LIN {X 0,Y 537.987,Z 364.092,A -85,B 0,C 180,E1 -4179.8,E2 -4179.8} C_VEL
LIN {X 0,Y 537.969,Z 364.095,A -85,B 0,C 180,E1 -4180.277,E2 -4180.277} C_VEL
LIN {X 0,Y 537.309,Z 364.183,A -85,B 0,C 180,E1 -4180.902,E2 -4180.902} C_VEL
LIN {X 0,Y 534.453,Z 364.538,A -85,B 0,C 180,E1 -4181.917,E2 -4181.917} C_VEL
LIN {X 0,Y 532.034,Z 364.837,A -85,B 0,C 180,E1 -4182.734,E2 -4182.734} C_VEL
LIN {X 0,Y 530.996,Z 364.964,A -85,B 0,C 180,E1 -4183.365,E2 -4183.365} C_VEL
LIN {X 0,Y 530.911,Z 364.973,A -85,B 0,C 180,E1 -4183.578,E2 -4183.578} C_VEL
LIN {X 0,Y 530.912,Z 364.974,A -85,B 0,C 180,E1 -4186.502,E2 -4186.502} C_VEL
LIN {X 0,Y 530.93,Z 364.969,A -85,B 0,C 180,E1 -4189.565,E2 -4189.565} C_VEL
LIN {X 0,Y 530.923,Z 364.975,A -85,B 0,C 180,E1 -4192.584,E2 -4192.584} C_VEL
LIN {X 0,Y 530.957,Z 364.96,A -85,B 0,C 180,E1 -4195.31,E2 -4195.31} C_VEL
LIN {X 0,Y 531.002,Z 365.136,A -85,B 0,C 180,E1 -4197.688,E2 -4197.688} C_VEL
LIN {X 0,Y 535.466,Z 381.503,A -85,B 0,C 180,E1 -4199.65,E2 -4199.65} C_VEL
LIN {X 0,Y 534.889,Z 405.466,A -85,B 0,C 180,E1 -4202.092,E2 -4202.092} C_VEL
LIN {X 0,Y 534.34,Z 429.212,A -85,B 0,C 180,E1 -4204.486,E2 -4204.486} C_VEL
LIN {X 0,Y 533.665,Z 459.976,A -85,B 0,C 180,E1 -4207.55,E2 -4207.55} C_VEL
LIN {X 0,Y 533.378,Z 473.259,A -85,B 0,C 180,E1 -4208.843,E2 -4208.843} C_VEL
LIN {X 0,Y 535.191,Z 484.127,A -85,B 0,C 180,E1 -4209.081,E2 -4209.081} C_VEL
LIN {X 0,Y 534.273,Z 640.741,A -85,B 0,C 180,E1 -4211.258,E2 -4211.258} C_VEL
LIN {X 0,Y 534.016,Z 655.888,A -85,B 0,C 180,E1 -4211.614,E2 -4211.614} C_VEL
LIN {X 0,Y 533.713,Z 669.614,A -85,B 0,C 180,E1 -4212.074,E2 -4212.074} C_VEL
LIN {X 0,Y 533.322,Z 682.934,A -85,B 0,C 180,E1 -4212.655,E2 -4212.655} C_VEL
LIN {X 0,Y 532.901,Z 696.987,A -85,B 0,C 180,E1 -4213.431,E2 -4213.431} C_VEL
LIN {X 0,Y 532.48,Z 710.223,A -85,B 0,C 180,E1 -4214.333,E2 -4214.333} C_VEL
LIN {X 0,Y 532.056,Z 722.77,A -85,B 0,C 180,E1 -4215.369,E2 -4215.369} C_VEL
LIN {X 0,Y 531.65,Z 733.601,A -85,B 0,C 180,E1 -4216.431,E2 -4216.431} C_VEL
LIN {X 0,Y 531.333,Z 743.593,A -85,B 0,C 180,E1 -4217.589,E2 -4217.589} C_VEL
LIN {X 0,Y 531.084,Z 753.363,A -85,B 0,C 180,E1 -4218.939,E2 -4218.939} C_VEL
LIN {X 0,Y 530.801,Z 761.478,A -85,B 0,C 180,E1 -4220.282,E2 -4220.282} C_VEL
LIN {X 0,Y 530.667,Z 768.204,A -85,B 0,C 180,E1 -4221.625,E2 -4221.625} C_VEL
LIN {X 0,Y 530.55,Z 774.441,A -85,B 0,C 180,E1 -4223.154,E2 -4223.154} C_VEL
LIN {X 0,Y 530.508,Z 779.264,A -85,B 0,C 180,E1 -4224.68,E2 -4224.68} C_VEL
LIN {X 0,Y 530.48,Z 782.801,A -85,B 0,C 180,E1 -4226.203,E2 -4226.203} C_VEL
LIN {X 0,Y 530.408,Z 785.143,A -85,B 0,C 180,E1 -4227.723,E2 -4227.723} C_VEL
LIN {X 0,Y 530.34,Z 786.339,A -85,B 0,C 180,E1 -4229.242,E2 -4229.242} C_VEL
LIN {X 0,Y 530.341,Z 786.358,A -85,B 0,C 180,E1 -4230.76,E2 -4230.76} C_VEL
LIN {X 0,Y 530.41,Z 785.237,A -85,B 0,C 180,E1 -4232.279,E2 -4232.279} C_VEL
LIN {X 0,Y 530.482,Z 782.969,A -85,B 0,C 180,E1 -4233.799,E2 -4233.799} C_VEL
LIN {X 0,Y 530.507,Z 779.504,A -85,B 0,C 180,E1 -4235.322,E2 -4235.322} C_VEL
LIN {X 0,Y 530.551,Z 774.76,A -85,B 0,C 180,E1 -4236.848,E2 -4236.848} C_VEL
LIN {X 0,Y 530.661,Z 768.615,A -85,B 0,C 180,E1 -4238.378,E2 -4238.378} C_VEL
LIN {X 0,Y 530.808,Z 760.885,A -85,B 0,C 180,E1 -4239.912,E2 -4239.912} C_VEL
LIN {X 0,Y 531.045,Z 752.644,A -85,B 0,C 180,E1 -4241.258,E2 -4241.258} C_VEL
LIN {X 0,Y 531.356,Z 742.721,A -85,B 0,C 180,E1 -4242.607,E2 -4242.607} C_VEL
LIN {X 0,Y 531.687,Z 732.601,A -85,B 0,C 180,E1 -4243.765,E2 -4243.765} C_VEL
LIN {X 0,Y 532.105,Z 720.489,A -85,B 0,C 180,E1 -4244.926,E2 -4244.926} C_VEL
LIN {X 0,Y 532.562,Z 708.684,A -85,B 0,C 180,E1 -4245.874,E2 -4245.874} C_VEL
LIN {X 0,Y 533.019,Z 695.268,A -85,B 0,C 180,E1 -4246.765,E2 -4246.765} C_VEL
LIN {X 0,Y 533.399,Z 680.725,A -85,B 0,C 180,E1 -4247.543,E2 -4247.543} C_VEL
LIN {X 0,Y 533.769,Z 666.821,A -85,B 0,C 180,E1 -4248.124,E2 -4248.124} C_VEL
LIN {X 0,Y 534.11,Z 651.426,A -85,B 0,C 180,E1 -4248.6,E2 -4248.6} C_VEL
LIN {X 0,Y 534.346,Z 635.503,A -85,B 0,C 180,E1 -4248.923,E2 -4248.923} C_VEL
LIN {X 0,Y 535.19,Z 484.115,A -85,B 0,C 180,E1 -4251.009,E2 -4251.009} C_VEL
LIN {X 0,Y 533.363,Z 472.907,A -85,B 0,C 180,E1 -4251.269,E2 -4251.269} C_VEL
LIN {X 0,Y 533.98,Z 444.484,A -85,B 0,C 180,E1 -4254.081,E2 -4254.081} C_VEL
LIN {X 0,Y 534.661,Z 417.063,A -85,B 0,C 180,E1 -4256.822,E2 -4256.822} C_VEL
LIN {X 0,Y 535.33,Z 389.185,A -85,B 0,C 180,E1 -4259.654,E2 -4259.654} C_VEL
LIN {X 0,Y 535.433,Z 381.261,A -85,B 0,C 180,E1 -4260.464,E2 -4260.464} C_VEL
LIN {X 0,Y 530.964,Z 365.143,A -85,B 0,C 180,E1 -4262.406,E2 -4262.406} C_VEL
LIN {X 0,Y 530.911,Z 364.972,A -85,B 0,C 180,E1 -4264.842,E2 -4264.842} C_VEL
LIN {X 0,Y 530.901,Z 364.981,A -85,B 0,C 180,E1 -4267.514,E2 -4267.514} C_VEL
LIN {X 0,Y 530.908,Z 364.975,A -85,B 0,C 180,E1 -4270.441,E2 -4270.441} C_VEL
LIN {X 0,Y 530.922,Z 364.977,A -85,B 0,C 180,E1 -4273.5,E2 -4273.5} C_VEL
LIN {X 0,Y 530.962,Z 364.966,A -85,B 0,C 180,E1 -4275.625,E2 -4275.625} C_VEL
LIN {X 0,Y 530.913,Z 364.975,A -85,B 0,C 180,E1 -4278.557,E2 -4278.557} C_VEL
LIN {X 0,Y 530.931,Z 364.975,A -85,B 0,C 180,E1 -4281.527,E2 -4281.527} C_VEL
LIN {X 0,Y 530.931,Z 364.967,A -85,B 0,C 180,E1 -4284.378,E2 -4284.378} C_VEL
LIN {X 0,Y 530.948,Z 364.972,A -85,B 0,C 180,E1 -4287.132,E2 -4287.132} C_VEL
LIN {X 0,Y 530.936,Z 364.971,A -85,B 0,C 180,E1 -4289.801,E2 -4289.801} C_VEL
LIN {X 0,Y 530.958,Z 364.969,A -85,B 0,C 180,E1 -4292.48,E2 -4292.48} C_VEL
LIN {X 0,Y 530.95,Z 364.971,A -85,B 0,C 180,E1 -4295.774,E2 -4295.774} C_VEL
LIN {X 0,Y 530.999,Z 364.97,A -85,B 0,C 180,E1 -4299.062,E2 -4299.062} C_VEL
LIN {X 0,Y 531.055,Z 365.122,A -85,B 0,C 180,E1 -4299.647,E2 -4299.647} C_VEL
LIN {X 0,Y 532.05,Z 371.983,A -85,B 0,C 180,E1 -4300.917,E2 -4300.917} C_VEL
LIN {X 0,Y 531.965,Z 377.818,A -85,B 0,C 180,E1 -4301.904,E2 -4301.904} C_VEL
LIN {X 0,Y 533.976,Z 387.187,A -85,B 0,C 180,E1 -4302.145,E2 -4302.145} C_VEL
LIN {X 0,Y 533.214,Z 515.389,A -85,B 0,C 180,E1 -4303.985,E2 -4303.985} C_VEL
LIN {X 0,Y 533.039,Z 529.891,A -85,B 0,C 180,E1 -4304.355,E2 -4304.355} C_VEL
LIN {X 0,Y 532.821,Z 543.338,A -85,B 0,C 180,E1 -4304.851,E2 -4304.851} C_VEL
LIN {X 0,Y 532.614,Z 556.223,A -85,B 0,C 180,E1 -4305.48,E2 -4305.48} C_VEL
LIN {X 0,Y 532.292,Z 567.295,A -85,B 0,C 180,E1 -4306.154,E2 -4306.154} C_VEL
LIN {X 0,Y 531.981,Z 578.921,A -85,B 0,C 180,E1 -4307.021,E2 -4307.021} C_VEL
LIN {X 0,Y 531.662,Z 589.877,A -85,B 0,C 180,E1 -4308.017,E2 -4308.017} C_VEL
LIN {X 0,Y 531.433,Z 599.998,A -85,B 0,C 180,E1 -4309.138,E2 -4309.138} C_VEL
LIN {X 0,Y 531.15,Z 608.633,A -85,B 0,C 180,E1 -4310.287,E2 -4310.287} C_VEL
LIN {X 0,Y 530.914,Z 616.868,A -85,B 0,C 180,E1 -4311.627,E2 -4311.627} C_VEL
LIN {X 0,Y 530.781,Z 622.612,A -85,B 0,C 180,E1 -4312.774,E2 -4312.774} C_VEL
LIN {X 0,Y 530.724,Z 628.655,A -85,B 0,C 180,E1 -4314.3,E2 -4314.3} C_VEL
LIN {X 0,Y 530.61,Z 632.169,A -85,B 0,C 180,E1 -4315.442,E2 -4315.442} C_VEL
LIN {X 0,Y 530.578,Z 635.531,A -85,B 0,C 180,E1 -4316.963,E2 -4316.963} C_VEL
LIN {X 0,Y 530.475,Z 637.559,A -85,B 0,C 180,E1 -4318.482,E2 -4318.482} C_VEL
LIN {X 0,Y 530.478,Z 638.29,A -85,B 0,C 180,E1 -4320,E2 -4320} C_VEL
LIN {X 0,Y 530.475,Z 637.723,A -85,B 0,C 180,E1 -4321.518,E2 -4321.518} C_VEL
LIN {X 0,Y 530.595,Z 635.831,A -85,B 0,C 180,E1 -4323.037,E2 -4323.037} C_VEL
LIN {X 0,Y 530.631,Z 632.609,A -85,B 0,C 180,E1 -4324.558,E2 -4324.558} C_VEL
LIN {X 0,Y 530.785,Z 627.929,A -85,B 0,C 180,E1 -4326.08,E2 -4326.08} C_VEL
LIN {X 0,Y 530.864,Z 621.641,A -85,B 0,C 180,E1 -4327.608,E2 -4327.608} C_VEL
LIN {X 0,Y 531.068,Z 614.585,A -85,B 0,C 180,E1 -4328.945,E2 -4328.945} C_VEL
LIN {X 0,Y 531.304,Z 605.793,A -85,B 0,C 180,E1 -4330.287,E2 -4330.287} C_VEL
LIN {X 0,Y 531.601,Z 596.53,A -85,B 0,C 180,E1 -4331.438,E2 -4331.438} C_VEL
LIN {X 0,Y 531.887,Z 586.212,A -85,B 0,C 180,E1 -4332.496,E2 -4332.496} C_VEL
LIN {X 0,Y 532.236,Z 574.76,A -85,B 0,C 180,E1 -4333.458,E2 -4333.458} C_VEL
LIN {X 0,Y 532.459,Z 563.55,A -85,B 0,C 180,E1 -4334.231,E2 -4334.231} C_VEL
LIN {X 0,Y 532.774,Z 551.386,A -85,B 0,C 180,E1 -4334.906,E2 -4334.906} C_VEL
LIN {X 0,Y 533.05,Z 539.454,A -85,B 0,C 180,E1 -4335.427,E2 -4335.427} C_VEL
LIN {X 0,Y 533.129,Z 525.988,A -85,B 0,C 180,E1 -4335.87,E2 -4335.87} C_VEL
LIN {X 0,Y 533.254,Z 510.983,A -85,B 0,C 180,E1 -4336.19,E2 -4336.19} C_VEL
LIN {X 0,Y 534.274,Z 387.61,A -85,B 0,C 180,E1 -4338.018,E2 -4338.018} C_VEL
LIN {X 0,Y 532.643,Z 380.641,A -85,B 0,C 180,E1 -4338.214,E2 -4338.214} C_VEL
LIN {X 0,Y 532.776,Z 373.678,A -85,B 0,C 180,E1 -4339.456,E2 -4339.456} C_VEL
LIN {X 0,Y 531.009,Z 365.099,A -85,B 0,C 180,E1 -4341.191,E2 -4341.191} C_VEL
LIN {X 0,Y 530.975,Z 364.971,A -85,B 0,C 180,E1 -4344.225,E2 -4344.225} C_VEL
LIN {X 0,Y 531.005,Z 364.969,A -85,B 0,C 180,E1 -4346.744,E2 -4346.744} C_VEL
LIN {X 0,Y 530.986,Z 364.967,A -85,B 0,C 180,E1 -4349.322,E2 -4349.322} C_VEL
LIN {X 0,Y 530.97,Z 364.971,A -85,B 0,C 180,E1 -4352.1,E2 -4352.1} C_VEL
LIN {X 0,Y 530.973,Z 364.971,A -85,B 0,C 180,E1 -4354.85,E2 -4354.85} C_VEL
LIN {X 0,Y 530.967,Z 364.968,A -85,B 0,C 180,E1 -4357.507,E2 -4357.507} C_VEL
LIN {X 0,Y 530.984,Z 364.972,A -85,B 0,C 180,E1 -4360.433,E2 -4360.433} C_VEL
LIN {X 0,Y 530.936,Z 364.971,A -85,B 0,C 180,E1 -4363.277,E2 -4363.277} C_VEL
LIN {X 0,Y 530.973,Z 364.969,A -85,B 0,C 180,E1 -4365.622,E2 -4365.622} C_VEL
LIN {X 0,Y 530.963,Z 364.972,A -85,B 0,C 180,E1 -4368.561,E2 -4368.561} C_VEL
LIN {X 0,Y 530.952,Z 364.973,A -85,B 0,C 180,E1 -4371.528,E2 -4371.528} C_VEL
LIN {X 0,Y 530.93,Z 364.977,A -85,B 0,C 180,E1 -4374.377,E2 -4374.377} C_VEL
LIN {X 0,Y 530.947,Z 364.974,A -85,B 0,C 180,E1 -4377.131,E2 -4377.131} C_VEL
LIN {X 0,Y 530.976,Z 365.169,A -85,B 0,C 180,E1 -4378.755,E2 -4378.755} C_VEL
LIN {X 0,Y 533.789,Z 375.588,A -85,B 0,C 180,E1 -4379.978,E2 -4379.978} C_VEL
LIN {X 0,Y 535.109,Z 381.227,A -85,B 0,C 180,E1 -4380.596,E2 -4380.596} C_VEL
LIN {X 0,Y 534.431,Z 411.488,A -85,B 0,C 180,E1 -4383.44,E2 -4383.44} C_VEL
LIN {X 0,Y 533.737,Z 445.316,A -85,B 0,C 180,E1 -4386.526,E2 -4386.526} C_VEL
LIN {X 0,Y 533.232,Z 471.07,A -85,B 0,C 180,E1 -4388.824,E2 -4388.824} C_VEL
LIN {X 0,Y 535.077,Z 484.407,A -85,B 0,C 180,E1 -4389.096,E2 -4389.096} C_VEL
LIN {X 0,Y 534.169,Z 640.097,A -85,B 0,C 180,E1 -4391.243,E2 -4391.243} C_VEL
LIN {X 0,Y 533.929,Z 655.851,A -85,B 0,C 180,E1 -4391.608,E2 -4391.608} C_VEL
LIN {X 0,Y 533.612,Z 671.04,A -85,B 0,C 180,E1 -4392.118,E2 -4392.118} C_VEL
LIN {X 0,Y 533.297,Z 685.298,A -85,B 0,C 180,E1 -4392.751,E2 -4392.751} C_VEL
LIN {X 0,Y 532.825,Z 699.152,A -85,B 0,C 180,E1 -4393.525,E2 -4393.525} C_VEL
LIN {X 0,Y 532.444,Z 711.668,A -85,B 0,C 180,E1 -4394.398,E2 -4394.398} C_VEL
LIN {X 0,Y 531.968,Z 724.282,A -85,B 0,C 180,E1 -4395.461,E2 -4395.461} C_VEL
LIN {X 0,Y 531.609,Z 735.737,A -85,B 0,C 180,E1 -4396.622,E2 -4396.622} C_VEL
LIN {X 0,Y 531.288,Z 745.38,A -85,B 0,C 180,E1 -4397.78,E2 -4397.78} C_VEL
LIN {X 0,Y 531.042,Z 754.844,A -85,B 0,C 180,E1 -4399.128,E2 -4399.128} C_VEL
LIN {X 0,Y 530.765,Z 762.723,A -85,B 0,C 180,E1 -4400.472,E2 -4400.472} C_VEL
LIN {X 0,Y 530.641,Z 770.083,A -85,B 0,C 180,E1 -4402.005,E2 -4402.005} C_VEL
LIN {X 0,Y 530.522,Z 775.774,A -85,B 0,C 180,E1 -4403.488,E2 -4403.488} C_VEL
LIN {X 0,Y 530.508,Z 779.383,A -85,B 0,C 180,E1 -4404.678,E2 -4404.678} C_VEL
LIN {X 0,Y 530.481,Z 782.881,A -85,B 0,C 180,E1 -4406.201,E2 -4406.201} C_VEL
LIN {X 0,Y 530.407,Z 785.185,A -85,B 0,C 180,E1 -4407.721,E2 -4407.721} C_VEL
LIN {X 0,Y 530.341,Z 786.347,A -85,B 0,C 180,E1 -4409.24,E2 -4409.24} C_VEL
LIN {X 0,Y 530.341,Z 786.348,A -85,B 0,C 180,E1 -4410.758,E2 -4410.758} C_VEL
LIN {X 0,Y 530.407,Z 785.191,A -85,B 0,C 180,E1 -4412.277,E2 -4412.277} C_VEL
LIN {X 0,Y 530.48,Z 782.889,A -85,B 0,C 180,E1 -4413.797,E2 -4413.797} C_VEL
LIN {X 0,Y 530.508,Z 779.389,A -85,B 0,C 180,E1 -4415.32,E2 -4415.32} C_VEL
LIN {X 0,Y 530.548,Z 774.61,A -85,B 0,C 180,E1 -4416.846,E2 -4416.846} C_VEL
LIN {X 0,Y 530.664,Z 768.428,A -85,B 0,C 180,E1 -4418.375,E2 -4418.375} C_VEL
LIN {X 0,Y 530.818,Z 760.655,A -85,B 0,C 180,E1 -4419.91,E2 -4419.91} C_VEL
LIN {X 0,Y 531.055,Z 752.376,A -85,B 0,C 180,E1 -4421.255,E2 -4421.255} C_VEL
LIN {X 0,Y 531.38,Z 742.401,A -85,B 0,C 180,E1 -4422.604,E2 -4422.604} C_VEL
LIN {X 0,Y 531.708,Z 732.196,A -85,B 0,C 180,E1 -4423.762,E2 -4423.762} C_VEL
LIN {X 0,Y 532.118,Z 720.025,A -85,B 0,C 180,E1 -4424.923,E2 -4424.923} C_VEL
LIN {X 0,Y 532.6,Z 706.602,A -85,B 0,C 180,E1 -4425.979,E2 -4425.979} C_VEL
LIN {X 0,Y 532.98,Z 694.363,A -85,B 0,C 180,E1 -4426.764,E2 -4426.764} C_VEL
LIN {X 0,Y 533.408,Z 679.29,A -85,B 0,C 180,E1 -4427.54,E2 -4427.54} C_VEL
LIN {X 0,Y 533.779,Z 664.666,A -85,B 0,C 180,E1 -4428.122,E2 -4428.122} C_VEL
LIN {X 0,Y 534.089,Z 648.748,A -85,B 0,C 180,E1 -4428.586,E2 -4428.586} C_VEL
LIN {X 0,Y 534.281,Z 632.911,A -85,B 0,C 180,E1 -4428.882,E2 -4428.882} C_VEL
LIN {X 0,Y 535.114,Z 484.112,A -85,B 0,C 180,E1 -4430.922,E2 -4430.922} C_VEL
LIN {X 0,Y 533.337,Z 471.527,A -85,B 0,C 180,E1 -4431.194,E2 -4431.194} C_VEL
LIN {X 0,Y 534.024,Z 441.043,A -85,B 0,C 180,E1 -4433.973,E2 -4433.973} C_VEL
LIN {X 0,Y 534.894,Z 407.916,A -85,B 0,C 180,E1 -4437.059,E2 -4437.059} C_VEL
LIN {X 0,Y 535.563,Z 383.049,A -85,B 0,C 180,E1 -4439.427,E2 -4439.427} C_VEL
LIN {X 0,Y 535.511,Z 381.106,A -85,B 0,C 180,E1 -4439.622,E2 -4439.622} C_VEL
LIN {X 0,Y 530.983,Z 365.172,A -85,B 0,C 180,E1 -4441.492,E2 -4441.492} C_VEL
LIN {X 0,Y 530.94,Z 364.976,A -85,B 0,C 180,E1 -4443.774,E2 -4443.774} C_VEL
LIN {X 0,Y 530.896,Z 364.98,A -85,B 0,C 180,E1 -4446.561,E2 -4446.561} C_VEL
LIN {X 0,Y 530.955,Z 364.969,A -85,B 0,C 180,E1 -4449.444,E2 -4449.444} C_VEL
LIN {X 0,Y 530.919,Z 364.98,A -85,B 0,C 180,E1 -4452.46,E2 -4452.46} C_VEL
LIN {X 0,Y 530.947,Z 364.968,A -85,B 0,C 180,E1 -4455.449,E2 -4455.449} C_VEL
LIN {X 0,Y 530.938,Z 364.967,A -85,B 0,C 180,E1 -4458.559,E2 -4458.559} C_VEL
LIN {X 0,Y 530.934,Z 364.97,A -85,B 0,C 180,E1 -4461.527,E2 -4461.527} C_VEL
LIN {X 0,Y 530.915,Z 364.964,A -85,B 0,C 180,E1 -4464.377,E2 -4464.377} C_VEL
LIN {X 0,Y 530.951,Z 364.967,A -85,B 0,C 180,E1 -4467.132,E2 -4467.132} C_VEL
LIN {X 0,Y 530.934,Z 364.971,A -85,B 0,C 180,E1 -4469.801,E2 -4469.801} C_VEL
LIN {X 0,Y 530.946,Z 364.977,A -85,B 0,C 180,E1 -4472.478,E2 -4472.478} C_VEL
LIN {X 0,Y 530.937,Z 364.967,A -85,B 0,C 180,E1 -4474.939,E2 -4474.939} C_VEL
LIN {X 0,Y 530.96,Z 364.968,A -85,B 0,C 180,E1 -4477.898,E2 -4477.898} C_VEL
LIN {X 0,Y 530.952,Z 364.973,A -85,B 0,C 180,E1 -4480.676,E2 -4480.676} C_VEL
LIN {X 0,Y 530.911,Z 364.973,A -85,B 0,C 180,E1 -4483.069,E2 -4483.069} C_VEL
LIN {X 0,Y 530.984,Z 364.959,A -85,B 0,C 180,E1 -4485.435,E2 -4485.435} C_VEL
LIN {X 0,Y 531.013,Z 364.966,A -85,B 0,C 180,E1 -4488.549,E2 -4488.549} C_VEL
LIN {X 0,Y 530.976,Z 364.962,A -85,B 0,C 180,E1 -4491.628,E2 -4491.628} C_VEL
LIN {X 0,Y 531.067,Z 364.955,A -85,B 0,C 180,E1 -4494.685,E2 -4494.685} C_VEL
LIN {X 0,Y 531.108,Z 364.947,A -85,B 0,C 180,E1 -4497.725,E2 -4497.725} C_VEL
LIN {X 0,Y 531.133,Z 364.946,A -85,B 0,C 180,E1 -4500.758,E2 -4500.758} C_VEL
LIN {X 0,Y 531.069,Z 364.956,A -85,B 0,C 180,E1 -4503.034,E2 -4503.034} C_VEL
LIN {X 0,Y 531.029,Z 364.958,A -85,B 0,C 180,E1 -4506.078,E2 -4506.078} C_VEL
LIN {X 0,Y 530.972,Z 364.968,A -85,B 0,C 180,E1 -4508.372,E2 -4508.372} C_VEL
LIN {X 0,Y 531.03,Z 364.952,A -85,B 0,C 180,E1 -4511.67,E2 -4511.67} C_VEL
LIN {X 0,Y 531.006,Z 364.963,A -85,B 0,C 180,E1 -4514.953,E2 -4514.953} C_VEL
LIN {X 0,Y 530.964,Z 364.964,A -85,B 0,C 180,E1 -4517.724,E2 -4517.724} C_VEL
LIN {X 0,Y 531.009,Z 364.961,A -85,B 0,C 180,E1 -4520.128,E2 -4520.128} C_VEL
LIN {X 0,Y 530.926,Z 364.976,A -85,B 0,C 180,E1 -4522.574,E2 -4522.574} C_VEL
LIN {X 0,Y 530.927,Z 364.972,A -85,B 0,C 180,E1 -4525.062,E2 -4525.062} C_VEL
LIN {X 0,Y 530.942,Z 364.969,A -85,B 0,C 180,E1 -4527.6,E2 -4527.6} C_VEL
LIN {X 0,Y 530.93,Z 364.977,A -85,B 0,C 180,E1 -4530.64,E2 -4530.64} C_VEL
LIN {X 0,Y 530.948,Z 364.969,A -85,B 0,C 180,E1 -4533.501,E2 -4533.501} C_VEL
LIN {X 0,Y 530.921,Z 364.972,A -85,B 0,C 180,E1 -4536.153,E2 -4536.153} C_VEL
LIN {X 0,Y 530.944,Z 364.968,A -85,B 0,C 180,E1 -4538.653,E2 -4538.653} C_VEL
LIN {X 0,Y 530.939,Z 364.967,A -85,B 0,C 180,E1 -4541.441,E2 -4541.441} C_VEL
LIN {X 0,Y 530.911,Z 364.973,A -85,B 0,C 180,E1 -4543.578,E2 -4543.578} C_VEL
LIN {X 0,Y 530.249,Z 365.057,A -85,B 0,C 180,E1 -4544.212,E2 -4544.212} C_VEL
LIN {X 0,Y 527.407,Z 365.412,A -85,B 0,C 180,E1 -4545.241,E2 -4545.241} C_VEL
LIN {X 0,Y 524.997,Z 365.712,A -85,B 0,C 180,E1 -4546.07,E2 -4546.07} C_VEL
LIN {X 0,Y 523.953,Z 365.84,A -85,B 0,C 180,E1 -4546.709,E2 -4546.709} C_VEL
LIN {X 0,Y 523.862,Z 365.851,A -85,B 0,C 180,E1 -4546.926,E2 -4546.926} C_VEL
LIN {X 0,Y 523.903,Z 365.844,A -85,B 0,C 180,E1 -4549.919,E2 -4549.919} C_VEL
LIN {X 0,Y 523.864,Z 365.852,A -85,B 0,C 180,E1 -4552.866,E2 -4552.866} C_VEL
LIN {X 0,Y 523.901,Z 365.832,A -85,B 0,C 180,E1 -4555.709,E2 -4555.709} C_VEL
LIN {X 0,Y 523.961,Z 366.063,A -85,B 0,C 180,E1 -4557.383,E2 -4557.383} C_VEL
LIN {X 0,Y 528.709,Z 383.052,A -85,B 0,C 180,E1 -4559.441,E2 -4559.441} C_VEL
LIN {X 0,Y 528.312,Z 403.383,A -85,B 0,C 180,E1 -4561.544,E2 -4561.544} C_VEL
LIN {X 0,Y 527.591,Z 429.824,A -85,B 0,C 180,E1 -4564.242,E2 -4564.242} C_VEL
LIN {X 0,Y 526.883,Z 458.525,A -85,B 0,C 180,E1 -4567.125,E2 -4567.125} C_VEL
LIN {X 0,Y 526.559,Z 472.845,A -85,B 0,C 180,E1 -4568.536,E2 -4568.536} C_VEL
LIN {X 0,Y 528.621,Z 486.323,A -85,B 0,C 180,E1 -4568.841,E2 -4568.841} C_VEL
LIN {X 0,Y 527.557,Z 640.53,A -85,B 0,C 180,E1 -4571.008,E2 -4571.008} C_VEL
LIN {X 0,Y 527.286,Z 655.836,A -85,B 0,C 180,E1 -4571.371,E2 -4571.371} C_VEL
LIN {X 0,Y 526.92,Z 670.811,A -85,B 0,C 180,E1 -4571.886,E2 -4571.886} C_VEL
LIN {X 0,Y 526.46,Z 684.812,A -85,B 0,C 180,E1 -4572.522,E2 -4572.522} C_VEL
LIN {X 0,Y 525.998,Z 698.494,A -85,B 0,C 180,E1 -4573.307,E2 -4573.307} C_VEL
LIN {X 0,Y 525.543,Z 711.522,A -85,B 0,C 180,E1 -4574.225,E2 -4574.225} C_VEL
LIN {X 0,Y 525.08,Z 723.802,A -85,B 0,C 180,E1 -4575.269,E2 -4575.269} C_VEL
LIN {X 0,Y 524.631,Z 735.342,A -85,B 0,C 180,E1 -4576.443,E2 -4576.443} C_VEL
LIN {X 0,Y 524.242,Z 746.435,A -85,B 0,C 180,E1 -4577.799,E2 -4577.799} C_VEL
LIN {X 0,Y 523.991,Z 755.799,A -85,B 0,C 180,E1 -4579.178,E2 -4579.178} C_VEL
LIN {X 0,Y 523.746,Z 762.523,A -85,B 0,C 180,E1 -4580.345,E2 -4580.345} C_VEL
LIN {X 0,Y 523.565,Z 769.921,A -85,B 0,C 180,E1 -4581.899,E2 -4581.899} C_VEL
LIN {X 0,Y 523.411,Z 776.044,A -85,B 0,C 180,E1 -4583.526,E2 -4583.526} C_VEL
LIN {X 0,Y 523.441,Z 779.265,A -85,B 0,C 180,E1 -4584.608,E2 -4584.608} C_VEL
LIN {X 0,Y 523.402,Z 782.802,A -85,B 0,C 180,E1 -4586.152,E2 -4586.152} C_VEL
LIN {X 0,Y 523.332,Z 785.143,A -85,B 0,C 180,E1 -4587.692,E2 -4587.692} C_VEL
LIN {X 0,Y 523.246,Z 786.339,A -85,B 0,C 180,E1 -4589.232,E2 -4589.232} C_VEL
LIN {X 0,Y 523.247,Z 786.358,A -85,B 0,C 180,E1 -4590.771,E2 -4590.771} C_VEL
LIN {X 0,Y 523.333,Z 785.237,A -85,B 0,C 180,E1 -4592.31,E2 -4592.31} C_VEL
LIN {X 0,Y 523.403,Z 782.968,A -85,B 0,C 180,E1 -4593.851,E2 -4593.851} C_VEL
LIN {X 0,Y 523.439,Z 779.502,A -85,B 0,C 180,E1 -4595.394,E2 -4595.394} C_VEL
LIN {X 0,Y 523.483,Z 774.756,A -85,B 0,C 180,E1 -4596.941,E2 -4596.941} C_VEL
LIN {X 0,Y 523.609,Z 768.61,A -85,B 0,C 180,E1 -4598.492,E2 -4598.492} C_VEL
LIN {X 0,Y 523.776,Z 760.88,A -85,B 0,C 180,E1 -4600.047,E2 -4600.047} C_VEL
LIN {X 0,Y 524.009,Z 752.637,A -85,B 0,C 180,E1 -4601.411,E2 -4601.411} C_VEL
LIN {X 0,Y 524.365,Z 742.711,A -85,B 0,C 180,E1 -4602.777,E2 -4602.777} C_VEL
LIN {X 0,Y 524.743,Z 732.583,A -85,B 0,C 180,E1 -4603.951,E2 -4603.951} C_VEL
LIN {X 0,Y 525.201,Z 720.559,A -85,B 0,C 180,E1 -4605.118,E2 -4605.118} C_VEL
LIN {X 0,Y 525.683,Z 708.377,A -85,B 0,C 180,E1 -4606.107,E2 -4606.107} C_VEL
LIN {X 0,Y 526.207,Z 695.221,A -85,B 0,C 180,E1 -4606.988,E2 -4606.988} C_VEL
LIN {X 0,Y 526.539,Z 682.661,A -85,B 0,C 180,E1 -4607.678,E2 -4607.678} C_VEL
LIN {X 0,Y 526.977,Z 668.007,A -85,B 0,C 180,E1 -4608.316,E2 -4608.316} C_VEL
LIN {X 0,Y 527.332,Z 652.493,A -85,B 0,C 180,E1 -4608.816,E2 -4608.816} C_VEL
LIN {X 0,Y 527.593,Z 637.697,A -85,B 0,C 180,E1 -4609.134,E2 -4609.134} C_VEL
LIN {X 0,Y 528.572,Z 485.348,A -85,B 0,C 180,E1 -4611.264,E2 -4611.264} C_VEL
LIN {X 0,Y 526.605,Z 473.206,A -85,B 0,C 180,E1 -4611.533,E2 -4611.533} C_VEL
LIN {X 0,Y 527.235,Z 444.14,A -85,B 0,C 180,E1 -4614.409,E2 -4614.409} C_VEL
LIN {X 0,Y 527.954,Z 416.184,A -85,B 0,C 180,E1 -4617.233,E2 -4617.233} C_VEL
LIN {X 0,Y 528.788,Z 386.926,A -85,B 0,C 180,E1 -4620.243,E2 -4620.243} C_VEL
LIN {X 0,Y 528.628,Z 382.804,A -85,B 0,C 180,E1 -4620.677,E2 -4620.677} C_VEL
LIN {X 0,Y 523.925,Z 366.076,A -85,B 0,C 180,E1 -4622.707,E2 -4622.707} C_VEL
LIN {X 0,Y 523.857,Z 365.835,A -85,B 0,C 180,E1 -4623.717,E2 -4623.717} C_VEL
LIN {X 0,Y 523.849,Z 365.854,A -85,B 0,C 180,E1 -4626.393,E2 -4626.393} C_VEL
LIN {X 0,Y 523.888,Z 365.85,A -85,B 0,C 180,E1 -4629.089,E2 -4629.089} C_VEL
LIN {X 0,Y 523.888,Z 365.843,A -85,B 0,C 180,E1 -4632.126,E2 -4632.126} C_VEL
LIN {X 0,Y 523.931,Z 365.842,A -85,B 0,C 180,E1 -4635.312,E2 -4635.312} C_VEL
LIN {X 0,Y 523.883,Z 365.852,A -85,B 0,C 180,E1 -4638.7,E2 -4638.7} C_VEL
LIN {X 0,Y 523.89,Z 365.849,A -85,B 0,C 180,E1 -4641.896,E2 -4641.896} C_VEL
LIN {X 0,Y 523.916,Z 365.841,A -85,B 0,C 180,E1 -4644.914,E2 -4644.914} C_VEL
LIN {X 0,Y 523.903,Z 365.848,A -85,B 0,C 180,E1 -4647.686,E2 -4647.686} C_VEL
LIN {X 0,Y 523.934,Z 365.845,A -85,B 0,C 180,E1 -4650.682,E2 -4650.682} C_VEL
LIN {X 0,Y 523.885,Z 365.851,A -85,B 0,C 180,E1 -4653.724,E2 -4653.724} C_VEL
LIN {X 0,Y 523.911,Z 365.847,A -85,B 0,C 180,E1 -4656.269,E2 -4656.269} C_VEL
LIN {X 0,Y 523.992,Z 365.907,A -85,B 0,C 180,E1 -4659.411,E2 -4659.411} C_VEL
LIN {X 0,Y 525.156,Z 373.557,A -85,B 0,C 180,E1 -4660.86,E2 -4660.86} C_VEL
LIN {X 0,Y 525.09,Z 378.407,A -85,B 0,C 180,E1 -4661.662,E2 -4661.662} C_VEL
LIN {X 0,Y 527.233,Z 388.321,A -85,B 0,C 180,E1 -4661.914,E2 -4661.914} C_VEL
LIN {X 0,Y 526.405,Z 516.027,A -85,B 0,C 180,E1 -4663.788,E2 -4663.788} C_VEL
LIN {X 0,Y 526.229,Z 530.054,A -85,B 0,C 180,E1 -4664.147,E2 -4664.147} C_VEL
LIN {X 0,Y 525.986,Z 543.668,A -85,B 0,C 180,E1 -4664.649,E2 -4664.649} C_VEL
LIN {X 0,Y 525.768,Z 556.66,A -85,B 0,C 180,E1 -4665.287,E2 -4665.287} C_VEL
LIN {X 0,Y 525.424,Z 567.816,A -85,B 0,C 180,E1 -4665.969,E2 -4665.969} C_VEL
LIN {X 0,Y 525.11,Z 579.51,A -85,B 0,C 180,E1 -4666.848,E2 -4666.848} C_VEL
LIN {X 0,Y 524.752,Z 590.726,A -85,B 0,C 180,E1 -4667.876,E2 -4667.876} C_VEL
LIN {X 0,Y 524.509,Z 600.721,A -85,B 0,C 180,E1 -4668.992,E2 -4668.992} C_VEL
LIN {X 0,Y 524.192,Z 609.405,A -85,B 0,C 180,E1 -4670.157,E2 -4670.157} C_VEL
LIN {X 0,Y 523.941,Z 617.704,A -85,B 0,C 180,E1 -4671.515,E2 -4671.515} C_VEL
LIN {X 0,Y 523.793,Z 623.469,A -85,B 0,C 180,E1 -4672.677,E2 -4672.677} C_VEL
LIN {X 0,Y 523.724,Z 629.574,A -85,B 0,C 180,E1 -4674.224,E2 -4674.224} C_VEL
LIN {X 0,Y 523.591,Z 633.102,A -85,B 0,C 180,E1 -4675.381,E2 -4675.381} C_VEL
LIN {X 0,Y 523.555,Z 636.516,A -85,B 0,C 180,E1 -4676.922,E2 -4676.922} C_VEL
LIN {X 0,Y 523.459,Z 638.568,A -85,B 0,C 180,E1 -4678.461,E2 -4678.461} C_VEL
LIN {X 0,Y 523.473,Z 639.314,A -85,B 0,C 180,E1 -4680,E2 -4680} C_VEL
LIN {X 0,Y 523.46,Z 638.762,A -85,B 0,C 180,E1 -4681.539,E2 -4681.539} C_VEL
LIN {X 0,Y 523.581,Z 636.878,A -85,B 0,C 180,E1 -4683.078,E2 -4683.078} C_VEL
LIN {X 0,Y 523.626,Z 633.656,A -85,B 0,C 180,E1 -4684.619,E2 -4684.619} C_VEL
LIN {X 0,Y 523.81,Z 628.953,A -85,B 0,C 180,E1 -4686.162,E2 -4686.162} C_VEL
LIN {X 0,Y 523.901,Z 622.648,A -85,B 0,C 180,E1 -4687.709,E2 -4687.709} C_VEL
LIN {X 0,Y 524.125,Z 615.572,A -85,B 0,C 180,E1 -4689.065,E2 -4689.065} C_VEL
LIN {X 0,Y 524.398,Z 606.739,A -85,B 0,C 180,E1 -4690.424,E2 -4690.424} C_VEL
LIN {X 0,Y 524.707,Z 597.421,A -85,B 0,C 180,E1 -4691.59,E2 -4691.59} C_VEL
LIN {X 0,Y 525.023,Z 587.051,A -85,B 0,C 180,E1 -4692.662,E2 -4692.662} C_VEL
LIN {X 0,Y 525.387,Z 575.533,A -85,B 0,C 180,E1 -4693.637,E2 -4693.637} C_VEL
LIN {X 0,Y 525.62,Z 564.24,A -85,B 0,C 180,E1 -4694.42,E2 -4694.42} C_VEL
LIN {X 0,Y 525.942,Z 551.965,A -85,B 0,C 180,E1 -4695.104,E2 -4695.104} C_VEL
LIN {X 0,Y 526.231,Z 538.953,A -85,B 0,C 180,E1 -4695.668,E2 -4695.668} C_VEL
LIN {X 0,Y 526.3,Z 525.252,A -85,B 0,C 180,E1 -4696.107,E2 -4696.107} C_VEL
LIN {X 0,Y 526.447,Z 510.738,A -85,B 0,C 180,E1 -4696.405,E2 -4696.405} C_VEL
LIN {X 0,Y 527.514,Z 399.224,A -85,B 0,C 180,E1 -4698.1,E2 -4698.1} C_VEL
LIN {X 0,Y 527.505,Z 387.848,A -85,B 0,C 180,E1 -4698.285,E2 -4698.285} C_VEL
LIN {X 0,Y 525.892,Z 381.547,A -85,B 0,C 180,E1 -4698.491,E2 -4698.491} C_VEL
LIN {X 0,Y 525.953,Z 374.776,A -85,B 0,C 180,E1 -4699.719,E2 -4699.719} C_VEL
LIN {X 0,Y 523.953,Z 365.886,A -85,B 0,C 180,E1 -4701.594,E2 -4701.594} C_VEL
LIN {X 0,Y 523.936,Z 365.849,A -85,B 0,C 180,E1 -4704.571,E2 -4704.571} C_VEL
LIN {X 0,Y 523.953,Z 365.846,A -85,B 0,C 180,E1 -4707.133,E2 -4707.133} C_VEL
LIN {X 0,Y 523.946,Z 365.844,A -85,B 0,C 180,E1 -4709.756,E2 -4709.756} C_VEL
LIN {X 0,Y 523.938,Z 365.85,A -85,B 0,C 180,E1 -4712.449,E2 -4712.449} C_VEL
LIN {X 0,Y 523.923,Z 365.846,A -85,B 0,C 180,E1 -4715.226,E2 -4715.226} C_VEL
LIN {X 0,Y 523.917,Z 365.85,A -85,B 0,C 180,E1 -4718.102,E2 -4718.102} C_VEL
LIN {X 0,Y 523.94,Z 365.844,A -85,B 0,C 180,E1 -4721.092,E2 -4721.092} C_VEL
LIN {X 0,Y 523.927,Z 365.851,A -85,B 0,C 180,E1 -4724.229,E2 -4724.229} C_VEL
LIN {X 0,Y 523.893,Z 365.851,A -85,B 0,C 180,E1 -4726.829,E2 -4726.829} C_VEL
LIN {X 0,Y 523.916,Z 365.852,A -85,B 0,C 180,E1 -4729.917,E2 -4729.917} C_VEL
LIN {X 0,Y 523.871,Z 365.853,A -85,B 0,C 180,E1 -4732.864,E2 -4732.864} C_VEL
LIN {X 0,Y 523.906,Z 365.853,A -85,B 0,C 180,E1 -4735.707,E2 -4735.707} C_VEL
LIN {X 0,Y 523.943,Z 366.048,A -85,B 0,C 180,E1 -4738.428,E2 -4738.428} C_VEL
LIN {X 0,Y 526.378,Z 374.842,A -85,B 0,C 180,E1 -4739.511,E2 -4739.511} C_VEL
LIN {X 0,Y 528.383,Z 382.678,A -85,B 0,C 180,E1 -4740.405,E2 -4740.405} C_VEL
LIN {X 0,Y 527.636,Z 411.618,A -85,B 0,C 180,E1 -4743.18,E2 -4743.18} C_VEL
LIN {X 0,Y 526.855,Z 444.151,A -85,B 0,C 180,E1 -4746.201,E2 -4746.201} C_VEL
LIN {X 0,Y 526.341,Z 469.965,A -85,B 0,C 180,E1 -4748.544,E2 -4748.544} C_VEL
LIN {X 0,Y 527.915,Z 481.484,A -85,B 0,C 180,E1 -4748.797,E2 -4748.797} C_VEL
LIN {X 0,Y 528.31,Z 486.446,A -85,B 0,C 180,E1 -4748.884,E2 -4748.884} C_VEL
LIN {X 0,Y 527.298,Z 639.796,A -85,B 0,C 180,E1 -4751.051,E2 -4751.051} C_VEL
LIN {X 0,Y 527.024,Z 655.705,A -85,B 0,C 180,E1 -4751.434,E2 -4751.434} C_VEL
LIN {X 0,Y 526.649,Z 671.244,A -85,B 0,C 180,E1 -4751.974,E2 -4751.974} C_VEL
LIN {X 0,Y 526.295,Z 685.289,A -85,B 0,C 180,E1 -4752.614,E2 -4752.614} C_VEL
LIN {X 0,Y 525.82,Z 699.081,A -85,B 0,C 180,E1 -4753.399,E2 -4753.399} C_VEL
LIN {X 0,Y 525.411,Z 713.14,A -85,B 0,C 180,E1 -4754.383,E2 -4754.383} C_VEL
LIN {X 0,Y 524.916,Z 725.845,A -85,B 0,C 180,E1 -4755.46,E2 -4755.46} C_VEL
LIN {X 0,Y 524.578,Z 737.389,A -85,B 0,C 180,E1 -4756.637,E2 -4756.637} C_VEL
LIN {X 0,Y 524.228,Z 746.867,A -85,B 0,C 180,E1 -4757.809,E2 -4757.809} C_VEL
LIN {X 0,Y 523.983,Z 756.073,A -85,B 0,C 180,E1 -4759.176,E2 -4759.176} C_VEL
LIN {X 0,Y 523.7,Z 764.737,A -85,B 0,C 180,E1 -4760.732,E2 -4760.732} C_VEL
LIN {X 0,Y 523.536,Z 771.696,A -85,B 0,C 180,E1 -4762.284,E2 -4762.284} C_VEL
LIN {X 0,Y 523.431,Z 777.162,A -85,B 0,C 180,E1 -4763.833,E2 -4763.833} C_VEL
LIN {X 0,Y 523.323,Z 781.285,A -85,B 0,C 180,E1 -4765.377,E2 -4765.377} C_VEL
LIN {X 0,Y 523.358,Z 784.177,A -85,B 0,C 180,E1 -4766.92,E2 -4766.92} C_VEL
LIN {X 0,Y 523.272,Z 785.906,A -85,B 0,C 180,E1 -4768.46,E2 -4768.46} C_VEL
LIN {X 0,Y 523.243,Z 786.5,A -85,B 0,C 180,E1 -4769.999,E2 -4769.999} C_VEL
LIN {X 0,Y 523.272,Z 785.91,A -85,B 0,C 180,E1 -4771.538,E2 -4771.538} C_VEL
LIN {X 0,Y 523.358,Z 784.186,A -85,B 0,C 180,E1 -4773.078,E2 -4773.078} C_VEL
LIN {X 0,Y 523.323,Z 781.293,A -85,B 0,C 180,E1 -4774.62,E2 -4774.62} C_VEL
LIN {X 0,Y 523.425,Z 777.165,A -85,B 0,C 180,E1 -4776.165,E2 -4776.165} C_VEL
LIN {X 0,Y 523.534,Z 771.704,A -85,B 0,C 180,E1 -4777.713,E2 -4777.713} C_VEL
LIN {X 0,Y 523.708,Z 764.755,A -85,B 0,C 180,E1 -4779.266,E2 -4779.266} C_VEL
LIN {X 0,Y 523.941,Z 757.305,A -85,B 0,C 180,E1 -4780.627,E2 -4780.627} C_VEL
LIN {X 0,Y 524.148,Z 748.269,A -85,B 0,C 180,E1 -4782.001,E2 -4782.001} C_VEL
LIN {X 0,Y 524.505,Z 739.076,A -85,B 0,C 180,E1 -4783.165,E2 -4783.165} C_VEL
LIN {X 0,Y 524.865,Z 727.934,A -85,B 0,C 180,E1 -4784.341,E2 -4784.341} C_VEL
LIN {X 0,Y 525.323,Z 715.158,A -85,B 0,C 180,E1 -4785.466,E2 -4785.466} C_VEL
LIN {X 0,Y 525.749,Z 702.397,A -85,B 0,C 180,E1 -4786.401,E2 -4786.401} C_VEL
LIN {X 0,Y 526.181,Z 689.456,A -85,B 0,C 180,E1 -4787.187,E2 -4787.187} C_VEL
LIN {X 0,Y 526.567,Z 675.462,A -85,B 0,C 180,E1 -4787.876,E2 -4787.876} C_VEL
LIN {X 0,Y 526.937,Z 660.632,A -85,B 0,C 180,E1 -4788.441,E2 -4788.441} C_VEL
LIN {X 0,Y 527.242,Z 645.419,A -85,B 0,C 180,E1 -4788.859,E2 -4788.859} C_VEL
LIN {X 0,Y 527.456,Z 628.131,A -85,B 0,C 180,E1 -4789.158,E2 -4789.158} C_VEL
LIN {X 0,Y 528.399,Z 484.563,A -85,B 0,C 180,E1 -4791.168,E2 -4791.168} C_VEL
LIN {X 0,Y 526.446,Z 471.328,A -85,B 0,C 180,E1 -4791.446,E2 -4791.446} C_VEL
LIN {X 0,Y 527.221,Z 441.531,A -85,B 0,C 180,E1 -4794.197,E2 -4794.197} C_VEL
LIN {X 0,Y 528.151,Z 408.395,A -85,B 0,C 180,E1 -4797.326,E2 -4797.326} C_VEL
LIN {X 0,Y 528.867,Z 383.46,A -85,B 0,C 180,E1 -4799.74,E2 -4799.74} C_VEL
LIN {X 0,Y 523.956,Z 366.061,A -85,B 0,C 180,E1 -4801.808,E2 -4801.808} C_VEL
LIN {X 0,Y 523.901,Z 365.853,A -85,B 0,C 180,E1 -4804.291,E2 -4804.291} C_VEL
LIN {X 0,Y 523.867,Z 365.854,A -85,B 0,C 180,E1 -4807.672,E2 -4807.672} C_VEL
LIN {X 0,Y 523.902,Z 365.853,A -85,B 0,C 180,E1 -4810.125,E2 -4810.125} C_VEL
LIN {X 0,Y 523.878,Z 365.85,A -85,B 0,C 180,E1 -4813.169,E2 -4813.169} C_VEL
LIN {X 0,Y 523.903,Z 365.848,A -85,B 0,C 180,E1 -4815.768,E2 -4815.768} C_VEL
LIN {X 0,Y 523.878,Z 365.847,A -85,B 0,C 180,E1 -4818.902,E2 -4818.902} C_VEL
LIN {X 0,Y 523.885,Z 365.851,A -85,B 0,C 180,E1 -4821.896,E2 -4821.896} C_VEL
LIN {X 0,Y 523.9,Z 365.835,A -85,B 0,C 180,E1 -4824.912,E2 -4824.912} C_VEL
LIN {X 0,Y 523.919,Z 365.843,A -85,B 0,C 180,E1 -4827.679,E2 -4827.679} C_VEL
LIN {X 0,Y 523.92,Z 365.846,A -85,B 0,C 180,E1 -4830.68,E2 -4830.68} C_VEL
LIN {X 0,Y 523.892,Z 365.848,A -85,B 0,C 180,E1 -4833.724,E2 -4833.724} C_VEL
LIN {X 0,Y 523.891,Z 365.849,A -85,B 0,C 180,E1 -4836.269,E2 -4836.269} C_VEL
LIN {X 0,Y 523.921,Z 365.845,A -85,B 0,C 180,E1 -4838.766,E2 -4838.766} C_VEL
LIN {X 0,Y 523.911,Z 365.844,A -85,B 0,C 180,E1 -4841.219,E2 -4841.219} C_VEL
LIN {X 0,Y 523.894,Z 365.85,A -85,B 0,C 180,E1 -4844.437,E2 -4844.437} C_VEL
LIN {X 0,Y 523.934,Z 365.842,A -85,B 0,C 180,E1 -4847.607,E2 -4847.607} C_VEL
LIN {X 0,Y 523.905,Z 365.844,A -85,B 0,C 180,E1 -4849.957,E2 -4849.957} C_VEL
LIN {X 0,Y 523.974,Z 365.838,A -85,B 0,C 180,E1 -4853.067,E2 -4853.067} C_VEL
LIN {X 0,Y 523.924,Z 365.837,A -85,B 0,C 180,E1 -4855.384,E2 -4855.384} C_VEL
LIN {X 0,Y 524.082,Z 365.822,A -85,B 0,C 180,E1 -4857.694,E2 -4857.694} C_VEL
LIN {X 0,Y 524.103,Z 365.821,A -85,B 0,C 180,E1 -4860.768,E2 -4860.768} C_VEL
LIN {X 0,Y 524.009,Z 365.835,A -85,B 0,C 180,E1 -4863.075,E2 -4863.075} C_VEL
LIN {X 0,Y 523.995,Z 365.835,A -85,B 0,C 180,E1 -4866.16,E2 -4866.16} C_VEL
LIN {X 0,Y 523.959,Z 365.839,A -85,B 0,C 180,E1 -4869.263,E2 -4869.263} C_VEL
LIN {X 0,Y 523.98,Z 365.83,A -85,B 0,C 180,E1 -4871.736,E2 -4871.736} C_VEL
LIN {X 0,Y 523.97,Z 365.838,A -85,B 0,C 180,E1 -4875.05,E2 -4875.05} C_VEL
LIN {X 0,Y 523.928,Z 365.841,A -85,B 0,C 180,E1 -4877.97,E2 -4877.97} C_VEL
LIN {X 0,Y 523.956,Z 365.843,A -85,B 0,C 180,E1 -4880.411,E2 -4880.411} C_VEL
LIN {X 0,Y 523.892,Z 365.853,A -85,B 0,C 180,E1 -4882.895,E2 -4882.895} C_VEL
LIN {X 0,Y 523.878,Z 365.846,A -85,B 0,C 180,E1 -4885.423,E2 -4885.423} C_VEL
LIN {X 0,Y 523.89,Z 365.848,A -85,B 0,C 180,E1 -4888.004,E2 -4888.004} C_VEL
LIN {X 0,Y 523.885,Z 365.856,A -85,B 0,C 180,E1 -4890.847,E2 -4890.847} C_VEL
LIN {X 0,Y 523.916,Z 365.845,A -85,B 0,C 180,E1 -4893.73,E2 -4893.73} C_VEL
LIN {X 0,Y 523.875,Z 365.852,A -85,B 0,C 180,E1 -4896.4,E2 -4896.4} C_VEL
LIN {X 0,Y 523.894,Z 365.852,A -85,B 0,C 180,E1 -4899.087,E2 -4899.087} C_VEL
LIN {X 0,Y 523.88,Z 365.846,A -85,B 0,C 180,E1 -4902.126,E2 -4902.126} C_VEL
LIN {X 0,Y 523.92,Z 365.845,A -85,B 0,C 180,E1 -4905.313,E2 -4905.313} C_VEL
LIN {X 0,Y 523.862,Z 365.851,A -85,B 0,C 180,E1 -4906.926,E2 -4906.926} C_VEL
LIN {X 0,Y 523.185,Z 365.938,A -85,B 0,C 180,E1 -4907.568,E2 -4907.568} C_VEL
LIN {X 0,Y 520.343,Z 366.296,A -85,B 0,C 180,E1 -4908.61,E2 -4908.61} C_VEL
LIN {X 0,Y 517.951,Z 366.589,A -85,B 0,C 180,E1 -4909.449,E2 -4909.449} C_VEL
LIN {X 0,Y 516.928,Z 366.713,A -85,B 0,C 180,E1 -4910.097,E2 -4910.097} C_VEL
LIN {X 0,Y 516.846,Z 366.723,A -85,B 0,C 180,E1 -4910.316,E2 -4910.316} C_VEL
LIN {X 0,Y 516.805,Z 366.731,A -85,B 0,C 180,E1 -4913.25,E2 -4913.25} C_VEL
LIN {X 0,Y 516.87,Z 366.7,A -85,B 0,C 180,E1 -4916.12,E2 -4916.12} C_VEL
LIN {X 0,Y 516.909,Z 366.93,A -85,B 0,C 180,E1 -4917.056,E2 -4917.056} C_VEL
LIN {X 0,Y 521.855,Z 384.559,A -85,B 0,C 180,E1 -4919.221,E2 -4919.221} C_VEL
LIN {X 0,Y 522.158,Z 386.811,A -85,B 0,C 180,E1 -4919.475,E2 -4919.475} C_VEL
LIN {X 0,Y 521.324,Z 414.907,A -85,B 0,C 180,E1 -4922.394,E2 -4922.394} C_VEL
LIN {X 0,Y 520.457,Z 443.906,A -85,B 0,C 180,E1 -4925.361,E2 -4925.361} C_VEL
LIN {X 0,Y 519.787,Z 472.76,A -85,B 0,C 180,E1 -4928.241,E2 -4928.241} C_VEL
LIN {X 0,Y 521.402,Z 482.574,A -85,B 0,C 180,E1 -4928.481,E2 -4928.481} C_VEL
LIN {X 0,Y 521.992,Z 487.311,A -85,B 0,C 180,E1 -4928.575,E2 -4928.575} C_VEL
LIN {X 0,Y 520.855,Z 640.508,A -85,B 0,C 180,E1 -4930.755,E2 -4930.755} C_VEL
LIN {X 0,Y 520.56,Z 655.774,A -85,B 0,C 180,E1 -4931.121,E2 -4931.121} C_VEL
LIN {X 0,Y 520.17,Z 670.765,A -85,B 0,C 180,E1 -4931.642,E2 -4931.642} C_VEL
LIN {X 0,Y 519.663,Z 684.776,A -85,B 0,C 180,E1 -4932.286,E2 -4932.286} C_VEL
LIN {X 0,Y 519.188,Z 698.466,A -85,B 0,C 180,E1 -4933.082,E2 -4933.082} C_VEL
LIN {X 0,Y 518.688,Z 711.189,A -85,B 0,C 180,E1 -4933.986,E2 -4933.986} C_VEL
LIN {X 0,Y 518.14,Z 723.783,A -85,B 0,C 180,E1 -4935.067,E2 -4935.067} C_VEL
LIN {X 0,Y 517.669,Z 735.325,A -85,B 0,C 180,E1 -4936.257,E2 -4936.257} C_VEL
LIN {X 0,Y 517.297,Z 745.056,A -85,B 0,C 180,E1 -4937.446,E2 -4937.446} C_VEL
LIN {X 0,Y 517.013,Z 754.58,A -85,B 0,C 180,E1 -4938.832,E2 -4938.832} C_VEL
LIN {X 0,Y 516.679,Z 762.517,A -85,B 0,C 180,E1 -4940.212,E2 -4940.212} C_VEL
LIN {X 0,Y 516.509,Z 769.919,A -85,B 0,C 180,E1 -4941.787,E2 -4941.787} C_VEL
LIN {X 0,Y 516.392,Z 774.443,A -85,B 0,C 180,E1 -4942.966,E2 -4942.966} C_VEL
LIN {X 0,Y 516.373,Z 779.266,A -85,B 0,C 180,E1 -4944.534,E2 -4944.534} C_VEL
LIN {X 0,Y 516.307,Z 782.803,A -85,B 0,C 180,E1 -4946.099,E2 -4946.099} C_VEL
LIN {X 0,Y 516.258,Z 785.143,A -85,B 0,C 180,E1 -4947.661,E2 -4947.661} C_VEL
LIN {X 0,Y 516.156,Z 786.339,A -85,B 0,C 180,E1 -4949.221,E2 -4949.221} C_VEL
LIN {X 0,Y 516.157,Z 786.358,A -85,B 0,C 180,E1 -4950.781,E2 -4950.781} C_VEL
LIN {X 0,Y 516.259,Z 785.236,A -85,B 0,C 180,E1 -4952.342,E2 -4952.342} C_VEL
LIN {X 0,Y 516.308,Z 782.967,A -85,B 0,C 180,E1 -4953.904,E2 -4953.904} C_VEL
LIN {X 0,Y 516.369,Z 779.499,A -85,B 0,C 180,E1 -4955.468,E2 -4955.468} C_VEL
LIN {X 0,Y 516.393,Z 774.753,A -85,B 0,C 180,E1 -4957.037,E2 -4957.037} C_VEL
LIN {X 0,Y 516.538,Z 768.603,A -85,B 0,C 180,E1 -4958.609,E2 -4958.609} C_VEL
LIN {X 0,Y 516.759,Z 760.866,A -85,B 0,C 180,E1 -4960.185,E2 -4960.185} C_VEL
LIN {X 0,Y 516.999,Z 752.617,A -85,B 0,C 180,E1 -4961.568,E2 -4961.568} C_VEL
LIN {X 0,Y 517.374,Z 742.685,A -85,B 0,C 180,E1 -4962.953,E2 -4962.953} C_VEL
LIN {X 0,Y 517.8,Z 732.554,A -85,B 0,C 180,E1 -4964.142,E2 -4964.142} C_VEL
LIN {X 0,Y 518.286,Z 720.89,A -85,B 0,C 180,E1 -4965.293,E2 -4965.293} C_VEL
LIN {X 0,Y 518.816,Z 708.604,A -85,B 0,C 180,E1 -4966.306,E2 -4966.306} C_VEL
LIN {X 0,Y 519.386,Z 695.171,A -85,B 0,C 180,E1 -4967.218,E2 -4967.218} C_VEL
LIN {X 0,Y 519.808,Z 681.642,A -85,B 0,C 180,E1 -4967.966,E2 -4967.966} C_VEL
LIN {X 0,Y 520.275,Z 666.663,A -85,B 0,C 180,E1 -4968.611,E2 -4968.611} C_VEL
LIN {X 0,Y 520.655,Z 651.332,A -85,B 0,C 180,E1 -4969.096,E2 -4969.096} C_VEL
LIN {X 0,Y 520.908,Z 636.825,A -85,B 0,C 180,E1 -4969.403,E2 -4969.403} C_VEL
LIN {X 0,Y 521.977,Z 486.695,A -85,B 0,C 180,E1 -4971.524,E2 -4971.524} C_VEL
LIN {X 0,Y 519.795,Z 473.141,A -85,B 0,C 180,E1 -4971.829,E2 -4971.829} C_VEL
LIN {X 0,Y 520.419,Z 445.801,A -85,B 0,C 180,E1 -4974.537,E2 -4974.537} C_VEL
LIN {X 0,Y 521.218,Z 417.781,A -85,B 0,C 180,E1 -4977.397,E2 -4977.397} C_VEL
LIN {X 0,Y 522.131,Z 387.766,A -85,B 0,C 180,E1 -4980.52,E2 -4980.52} C_VEL
LIN {X 0,Y 521.81,Z 384.333,A -85,B 0,C 180,E1 -4980.897,E2 -4980.897} C_VEL
LIN {X 0,Y 516.88,Z 366.94,A -85,B 0,C 180,E1 -4983.036,E2 -4983.036} C_VEL
LIN {X 0,Y 516.826,Z 366.725,A -85,B 0,C 180,E1 -4984.83,E2 -4984.83} C_VEL
LIN {X 0,Y 516.835,Z 366.73,A -85,B 0,C 180,E1 -4987.936,E2 -4987.936} C_VEL
LIN {X 0,Y 516.823,Z 366.733,A -85,B 0,C 180,E1 -4990.748,E2 -4990.748} C_VEL
LIN {X 0,Y 516.863,Z 366.725,A -85,B 0,C 180,E1 -4993.906,E2 -4993.906} C_VEL
LIN {X 0,Y 516.863,Z 366.719,A -85,B 0,C 180,E1 -4996.11,E2 -4996.11} C_VEL
LIN {X 0,Y 516.826,Z 366.725,A -85,B 0,C 180,E1 -4999.253,E2 -4999.253} C_VEL
LIN {X 0,Y 516.853,Z 366.725,A -85,B 0,C 180,E1 -5002.062,E2 -5002.062} C_VEL
LIN {X 0,Y 516.871,Z 366.717,A -85,B 0,C 180,E1 -5005.174,E2 -5005.174} C_VEL
LIN {X 0,Y 516.849,Z 366.725,A -85,B 0,C 180,E1 -5007.973,E2 -5007.973} C_VEL
LIN {X 0,Y 516.902,Z 366.722,A -85,B 0,C 180,E1 -5010.694,E2 -5010.694} C_VEL
LIN {X 0,Y 516.862,Z 366.726,A -85,B 0,C 180,E1 -5013.824,E2 -5013.824} C_VEL
LIN {X 0,Y 516.859,Z 366.729,A -85,B 0,C 180,E1 -5016.776,E2 -5016.776} C_VEL
LIN {X 0,Y 516.97,Z 366.89,A -85,B 0,C 180,E1 -5019.249,E2 -5019.249} C_VEL
LIN {X 0,Y 518.248,Z 374.026,A -85,B 0,C 180,E1 -5020.595,E2 -5020.595} C_VEL
LIN {X 0,Y 518.229,Z 378.879,A -85,B 0,C 180,E1 -5021.405,E2 -5021.405} C_VEL
LIN {X 0,Y 520.533,Z 389.471,A -85,B 0,C 180,E1 -5021.678,E2 -5021.678} C_VEL
LIN {X 0,Y 519.582,Z 516.128,A -85,B 0,C 180,E1 -5023.573,E2 -5023.573} C_VEL
LIN {X 0,Y 519.411,Z 529.966,A -85,B 0,C 180,E1 -5023.925,E2 -5023.925} C_VEL
LIN {X 0,Y 519.167,Z 543.993,A -85,B 0,C 180,E1 -5024.443,E2 -5024.443} C_VEL
LIN {X 0,Y 518.93,Z 557.093,A -85,B 0,C 180,E1 -5025.089,E2 -5025.089} C_VEL
LIN {X 0,Y 518.551,Z 568.336,A -85,B 0,C 180,E1 -5025.78,E2 -5025.78} C_VEL
LIN {X 0,Y 518.234,Z 580.101,A -85,B 0,C 180,E1 -5026.671,E2 -5026.671} C_VEL
LIN {X 0,Y 517.833,Z 591.639,A -85,B 0,C 180,E1 -5027.738,E2 -5027.738} C_VEL
LIN {X 0,Y 517.588,Z 601.445,A -85,B 0,C 180,E1 -5028.843,E2 -5028.843} C_VEL
LIN {X 0,Y 517.241,Z 610.177,A -85,B 0,C 180,E1 -5030.024,E2 -5030.024} C_VEL
LIN {X 0,Y 516.974,Z 618.528,A -85,B 0,C 180,E1 -5031.4,E2 -5031.4} C_VEL
LIN {X 0,Y 516.812,Z 624.325,A -85,B 0,C 180,E1 -5032.577,E2 -5032.577} C_VEL
LIN {X 0,Y 516.749,Z 629.087,A -85,B 0,C 180,E1 -5033.754,E2 -5033.754} C_VEL
LIN {X 0,Y 516.575,Z 634.033,A -85,B 0,C 180,E1 -5035.318,E2 -5035.318} C_VEL
LIN {X 0,Y 516.531,Z 637.491,A -85,B 0,C 180,E1 -5036.88,E2 -5036.88} C_VEL
LIN {X 0,Y 516.444,Z 639.576,A -85,B 0,C 180,E1 -5038.44,E2 -5038.44} C_VEL
LIN {X 0,Y 516.467,Z 640.338,A -85,B 0,C 180,E1 -5040,E2 -5040} C_VEL
LIN {X 0,Y 516.444,Z 639.802,A -85,B 0,C 180,E1 -5041.56,E2 -5041.56} C_VEL
LIN {X 0,Y 516.568,Z 637.924,A -85,B 0,C 180,E1 -5043.12,E2 -5043.12} C_VEL
LIN {X 0,Y 516.621,Z 634.695,A -85,B 0,C 180,E1 -5044.682,E2 -5044.682} C_VEL
LIN {X 0,Y 516.835,Z 629.978,A -85,B 0,C 180,E1 -5046.245,E2 -5046.245} C_VEL
LIN {X 0,Y 516.867,Z 625.411,A -85,B 0,C 180,E1 -5047.422,E2 -5047.422} C_VEL
LIN {X 0,Y 517.113,Z 618.726,A -85,B 0,C 180,E1 -5048.795,E2 -5048.795} C_VEL
LIN {X 0,Y 517.353,Z 610.397,A -85,B 0,C 180,E1 -5050.172,E2 -5050.172} C_VEL
LIN {X 0,Y 517.735,Z 601.624,A -85,B 0,C 180,E1 -5051.352,E2 -5051.352} C_VEL
LIN {X 0,Y 518.041,Z 592.585,A -85,B 0,C 180,E1 -5052.367,E2 -5052.367} C_VEL
LIN {X 0,Y 518.382,Z 581.235,A -85,B 0,C 180,E1 -5053.425,E2 -5053.425} C_VEL
LIN {X 0,Y 518.667,Z 569.497,A -85,B 0,C 180,E1 -5054.317,E2 -5054.317} C_VEL
LIN {X 0,Y 519.012,Z 556.459,A -85,B 0,C 180,E1 -5055.11,E2 -5055.11} C_VEL
LIN {X 0,Y 519.36,Z 542.602,A -85,B 0,C 180,E1 -5055.754,E2 -5055.754} C_VEL
LIN {X 0,Y 519.501,Z 528.383,A -85,B 0,C 180,E1 -5056.243,E2 -5056.243} C_VEL
LIN {X 0,Y 519.617,Z 514.906,A -85,B 0,C 180,E1 -5056.551,E2 -5056.551} C_VEL
LIN {X 0,Y 520.959,Z 394.609,A -85,B 0,C 180,E1 -5058.447,E2 -5058.447} C_VEL
LIN {X 0,Y 520.925,Z 389.155,A -85,B 0,C 180,E1 -5058.542,E2 -5058.542} C_VEL
LIN {X 0,Y 519.202,Z 382.802,A -85,B 0,C 180,E1 -5058.747,E2 -5058.747} C_VEL
LIN {X 0,Y 519.196,Z 380.238,A -85,B 0,C 180,E1 -5059.163,E2 -5059.163} C_VEL
LIN {X 0,Y 519.222,Z 377.012,A -85,B 0,C 180,E1 -5059.779,E2 -5059.779} C_VEL
LIN {X 0,Y 516.914,Z 366.783,A -85,B 0,C 180,E1 -5061.956,E2 -5061.956} C_VEL
LIN {X 0,Y 516.913,Z 366.725,A -85,B 0,C 180,E1 -5064.928,E2 -5064.928} C_VEL
LIN {X 0,Y 516.929,Z 366.718,A -85,B 0,C 180,E1 -5067.905,E2 -5067.905} C_VEL
LIN {X 0,Y 516.896,Z 366.725,A -85,B 0,C 180,E1 -5070.203,E2 -5070.203} C_VEL
LIN {X 0,Y 516.899,Z 366.724,A -85,B 0,C 180,E1 -5072.947,E2 -5072.947} C_VEL
LIN {X 0,Y 516.872,Z 366.725,A -85,B 0,C 180,E1 -5075.78,E2 -5075.78} C_VEL
LIN {X 0,Y 516.883,Z 366.727,A -85,B 0,C 180,E1 -5078.716,E2 -5078.716} C_VEL
LIN {X 0,Y 516.91,Z 366.721,A -85,B 0,C 180,E1 -5081.775,E2 -5081.775} C_VEL
LIN {X 0,Y 516.899,Z 366.721,A -85,B 0,C 180,E1 -5085.006,E2 -5085.006} C_VEL
LIN {X 0,Y 516.889,Z 366.727,A -85,B 0,C 180,E1 -5088.402,E2 -5088.402} C_VEL
LIN {X 0,Y 516.876,Z 366.725,A -85,B 0,C 180,E1 -5091.283,E2 -5091.283} C_VEL
LIN {X 0,Y 516.851,Z 366.73,A -85,B 0,C 180,E1 -5094.673,E2 -5094.673} C_VEL
LIN {X 0,Y 516.866,Z 366.731,A -85,B 0,C 180,E1 -5097.462,E2 -5097.462} C_VEL
LIN {X 0,Y 516.941,Z 367.015,A -85,B 0,C 180,E1 -5098.114,E2 -5098.114} C_VEL
LIN {X 0,Y 520.61,Z 380.428,A -85,B 0,C 180,E1 -5099.765,E2 -5099.765} C_VEL
LIN {X 0,Y 521.681,Z 385.323,A -85,B 0,C 180,E1 -5100.323,E2 -5100.323} C_VEL
LIN {X 0,Y 520.727,Z 415.18,A -85,B 0,C 180,E1 -5103.239,E2 -5103.239} C_VEL
LIN {X 0,Y 519.897,Z 447.479,A -85,B 0,C 180,E1 -5106.286,E2 -5106.286} C_VEL
LIN {X 0,Y 519.433,Z 468.683,A -85,B 0,C 180,E1 -5108.244,E2 -5108.244} C_VEL
LIN {X 0,Y 519.637,Z 471.47,A -85,B 0,C 180,E1 -5108.337,E2 -5108.337} C_VEL
LIN {X 0,Y 521.585,Z 485.107,A -85,B 0,C 180,E1 -5108.621,E2 -5108.621} C_VEL
LIN {X 0,Y 520.564,Z 625.404,A -85,B 0,C 180,E1 -5110.633,E2 -5110.633} C_VEL
LIN {X 0,Y 520.331,Z 643.116,A -85,B 0,C 180,E1 -5110.931,E2 -5110.931} C_VEL
LIN {X 0,Y 520.018,Z 658.674,A -85,B 0,C 180,E1 -5111.353,E2 -5111.353} C_VEL
LIN {X 0,Y 519.612,Z 673.76,A -85,B 0,C 180,E1 -5111.925,E2 -5111.925} C_VEL
LIN {X 0,Y 519.263,Z 687.042,A -85,B 0,C 180,E1 -5112.574,E2 -5112.574} C_VEL
LIN {X 0,Y 518.713,Z 701.806,A -85,B 0,C 180,E1 -5113.468,E2 -5113.468} C_VEL
LIN {X 0,Y 518.241,Z 714.906,A -85,B 0,C 180,E1 -5114.441,E2 -5114.441} C_VEL
LIN {X 0,Y 517.793,Z 727.413,A -85,B 0,C 180,E1 -5115.557,E2 -5115.557} C_VEL
LIN {X 0,Y 517.397,Z 739.457,A -85,B 0,C 180,E1 -5116.848,E2 -5116.848} C_VEL
LIN {X 0,Y 517.008,Z 750.203,A -85,B 0,C 180,E1 -5118.234,E2 -5118.234} C_VEL
LIN {X 0,Y 516.803,Z 759.139,A -85,B 0,C 180,E1 -5119.618,E2 -5119.618} C_VEL
LIN {X 0,Y 516.589,Z 766.501,A -85,B 0,C 180,E1 -5120.998,E2 -5120.998} C_VEL
LIN {X 0,Y 516.43,Z 773.179,A -85,B 0,C 180,E1 -5122.571,E2 -5122.571} C_VEL
LIN {X 0,Y 516.373,Z 778.319,A -85,B 0,C 180,E1 -5124.14,E2 -5124.14} C_VEL
LIN {X 0,Y 516.239,Z 781.285,A -85,B 0,C 180,E1 -5125.314,E2 -5125.314} C_VEL
LIN {X 0,Y 516.272,Z 784.176,A -85,B 0,C 180,E1 -5126.877,E2 -5126.877} C_VEL
LIN {X 0,Y 516.189,Z 785.905,A -85,B 0,C 180,E1 -5128.438,E2 -5128.438} C_VEL
LIN {X 0,Y 516.151,Z 786.5,A -85,B 0,C 180,E1 -5129.999,E2 -5129.999} C_VEL
LIN {X 0,Y 516.189,Z 785.909,A -85,B 0,C 180,E1 -5131.559,E2 -5131.559} C_VEL
LIN {X 0,Y 516.271,Z 784.185,A -85,B 0,C 180,E1 -5133.12,E2 -5133.12} C_VEL
LIN {X 0,Y 516.238,Z 781.292,A -85,B 0,C 180,E1 -5134.684,E2 -5134.684} C_VEL
LIN {X 0,Y 516.371,Z 778.324,A -85,B 0,C 180,E1 -5135.858,E2 -5135.858} C_VEL
LIN {X 0,Y 516.428,Z 773.186,A -85,B 0,C 180,E1 -5137.427,E2 -5137.427} C_VEL
LIN {X 0,Y 516.59,Z 766.519,A -85,B 0,C 180,E1 -5139,E2 -5139} C_VEL
LIN {X 0,Y 516.802,Z 759.177,A -85,B 0,C 180,E1 -5140.379,E2 -5140.379} C_VEL
LIN {X 0,Y 517.023,Z 749.748,A -85,B 0,C 180,E1 -5141.844,E2 -5141.844} C_VEL
LIN {X 0,Y 517.394,Z 739.673,A -85,B 0,C 180,E1 -5143.15,E2 -5143.15} C_VEL
LIN {X 0,Y 517.818,Z 727.768,A -85,B 0,C 180,E1 -5144.44,E2 -5144.44} C_VEL
LIN {X 0,Y 518.293,Z 715.14,A -85,B 0,C 180,E1 -5145.58,E2 -5145.58} C_VEL
LIN {X 0,Y 518.763,Z 702.544,A -85,B 0,C 180,E1 -5146.527,E2 -5146.527} C_VEL
LIN {X 0,Y 519.204,Z 689.833,A -85,B 0,C 180,E1 -5147.324,E2 -5147.324} C_VEL
LIN {X 0,Y 519.633,Z 676.178,A -85,B 0,C 180,E1 -5148.021,E2 -5148.021} C_VEL
LIN {X 0,Y 520.039,Z 661.104,A -85,B 0,C 180,E1 -5148.618,E2 -5148.618} C_VEL
LIN {X 0,Y 520.39,Z 645.945,A -85,B 0,C 180,E1 -5149.054,E2 -5149.054} C_VEL
LIN {X 0,Y 520.639,Z 629.443,A -85,B 0,C 180,E1 -5149.355,E2 -5149.355} C_VEL
LIN {X 0,Y 521.732,Z 485.613,A -85,B 0,C 180,E1 -5151.41,E2 -5151.41} C_VEL
LIN {X 0,Y 519.62,Z 470.499,A -85,B 0,C 180,E1 -5151.741,E2 -5151.741} C_VEL
LIN {X 0,Y 520.512,Z 438.71,A -85,B 0,C 180,E1 -5154.742,E2 -5154.742} C_VEL
LIN {X 0,Y 521.529,Z 405.556,A -85,B 0,C 180,E1 -5157.921,E2 -5157.921} C_VEL
LIN {X 0,Y 522.227,Z 385.809,A -85,B 0,C 180,E1 -5159.862,E2 -5159.862} C_VEL
LIN {X 0,Y 517.759,Z 369.975,A -85,B 0,C 180,E1 -5161.739,E2 -5161.739} C_VEL
LIN {X 0,Y 516.917,Z 366.88,A -85,B 0,C 180,E1 -5162.154,E2 -5162.154} C_VEL
LIN {X 0,Y 516.86,Z 366.728,A -85,B 0,C 180,E1 -5164.825,E2 -5164.825} C_VEL
LIN {X 0,Y 516.849,Z 366.731,A -85,B 0,C 180,E1 -5167.939,E2 -5167.939} C_VEL
LIN {X 0,Y 516.841,Z 366.73,A -85,B 0,C 180,E1 -5170.744,E2 -5170.744} C_VEL
LIN {X 0,Y 516.869,Z 366.726,A -85,B 0,C 180,E1 -5173.902,E2 -5173.902} C_VEL
LIN {X 0,Y 516.846,Z 366.728,A -85,B 0,C 180,E1 -5176.109,E2 -5176.109} C_VEL
LIN {X 0,Y 516.836,Z 366.722,A -85,B 0,C 180,E1 -5179.254,E2 -5179.254} C_VEL
LIN {X 0,Y 516.845,Z 366.73,A -85,B 0,C 180,E1 -5182.059,E2 -5182.059} C_VEL
LIN {X 0,Y 516.856,Z 366.71,A -85,B 0,C 180,E1 -5185.173,E2 -5185.173} C_VEL
LIN {X 0,Y 516.856,Z 366.725,A -85,B 0,C 180,E1 -5187.974,E2 -5187.974} C_VEL
LIN {X 0,Y 516.888,Z 366.721,A -85,B 0,C 180,E1 -5190.693,E2 -5190.693} C_VEL
LIN {X 0,Y 516.871,Z 366.723,A -85,B 0,C 180,E1 -5193.816,E2 -5193.816} C_VEL
LIN {X 0,Y 516.84,Z 366.73,A -85,B 0,C 180,E1 -5196.775,E2 -5196.775} C_VEL
LIN {X 0,Y 516.911,Z 366.714,A -85,B 0,C 180,E1 -5199.735,E2 -5199.735} C_VEL
LIN {X 0,Y 516.848,Z 366.731,A -85,B 0,C 180,E1 -5202.593,E2 -5202.593} C_VEL
LIN {X 0,Y 516.915,Z 366.713,A -85,B 0,C 180,E1 -5205.029,E2 -5205.029} C_VEL
LIN {X 0,Y 516.95,Z 366.717,A -85,B 0,C 180,E1 -5208.233,E2 -5208.233} C_VEL
LIN {X 0,Y 516.908,Z 366.714,A -85,B 0,C 180,E1 -5211.399,E2 -5211.399} C_VEL
LIN {X 0,Y 516.963,Z 366.713,A -85,B 0,C 180,E1 -5214.539,E2 -5214.539} C_VEL
LIN {X 0,Y 517.054,Z 366.698,A -85,B 0,C 180,E1 -5217.663,E2 -5217.663} C_VEL
LIN {X 0,Y 517.073,Z 366.696,A -85,B 0,C 180,E1 -5220.779,E2 -5220.779} C_VEL
LIN {X 0,Y 516.95,Z 366.714,A -85,B 0,C 180,E1 -5223.117,E2 -5223.117} C_VEL
LIN {X 0,Y 516.964,Z 366.711,A -85,B 0,C 180,E1 -5226.244,E2 -5226.244} C_VEL
LIN {X 0,Y 516.915,Z 366.716,A -85,B 0,C 180,E1 -5229.39,E2 -5229.39} C_VEL
LIN {X 0,Y 516.936,Z 366.707,A -85,B 0,C 180,E1 -5231.807,E2 -5231.807} C_VEL
LIN {X 0,Y 516.923,Z 366.715,A -85,B 0,C 180,E1 -5235.144,E2 -5235.144} C_VEL
LIN {X 0,Y 516.896,Z 366.719,A -85,B 0,C 180,E1 -5238.223,E2 -5238.223} C_VEL
LIN {X 0,Y 516.896,Z 366.721,A -85,B 0,C 180,E1 -5240.702,E2 -5240.702} C_VEL
LIN {X 0,Y 516.868,Z 366.724,A -85,B 0,C 180,E1 -5244.074,E2 -5244.074} C_VEL
LIN {X 0,Y 516.819,Z 366.734,A -85,B 0,C 180,E1 -5246.664,E2 -5246.664} C_VEL
LIN {X 0,Y 516.865,Z 366.721,A -85,B 0,C 180,E1 -5249.518,E2 -5249.518} C_VEL
LIN {X 0,Y 516.866,Z 366.728,A -85,B 0,C 180,E1 -5252.949,E2 -5252.949} C_VEL
LIN {X 0,Y 516.85,Z 366.723,A -85,B 0,C 180,E1 -5255.782,E2 -5255.782} C_VEL
LIN {X 0,Y 516.858,Z 366.722,A -85,B 0,C 180,E1 -5258.718,E2 -5258.718} C_VEL
LIN {X 0,Y 516.832,Z 366.722,A -85,B 0,C 180,E1 -5261.783,E2 -5261.783} C_VEL
LIN {X 0,Y 516.885,Z 366.726,A -85,B 0,C 180,E1 -5265.008,E2 -5265.008} C_VEL
LIN {X 0,Y 516.838,Z 366.73,A -85,B 0,C 180,E1 -5268.408,E2 -5268.408} C_VEL
LIN {X 0,Y 516.846,Z 366.723,A -85,B 0,C 180,E1 -5270.316,E2 -5270.316} C_VEL
LIN {X 0,Y 516.18,Z 366.813,A -85,B 0,C 180,E1 -5270.966,E2 -5270.966} C_VEL
LIN {X 0,Y 513.311,Z 367.169,A -85,B 0,C 180,E1 -5272.022,E2 -5272.022} C_VEL
LIN {X 0,Y 510.885,Z 367.472,A -85,B 0,C 180,E1 -5272.872,E2 -5272.872} C_VEL
LIN {X 0,Y 509.843,Z 367.601,A -85,B 0,C 180,E1 -5273.529,E2 -5273.529} C_VEL
LIN {X 0,Y 509.759,Z 367.612,A -85,B 0,C 180,E1 -5273.751,E2 -5273.751} C_VEL
LIN {X 0,Y 509.862,Z 367.673,A -85,B 0,C 180,E1 -5276.676,E2 -5276.676} C_VEL
LIN {X 0,Y 510.227,Z 369.132,A -85,B 0,C 180,E1 -5276.915,E2 -5276.915} C_VEL
LIN {X 0,Y 514.983,Z 385.82,A -85,B 0,C 180,E1 -5278.967,E2 -5278.967} C_VEL
LIN {X 0,Y 515.461,Z 388.928,A -85,B 0,C 180,E1 -5279.327,E2 -5279.327} C_VEL
LIN {X 0,Y 514.501,Z 420.206,A -85,B 0,C 180,E1 -5282.609,E2 -5282.609} C_VEL
LIN {X 0,Y 513.504,Z 451.879,A -85,B 0,C 180,E1 -5285.867,E2 -5285.867} C_VEL
LIN {X 0,Y 513,Z 472.884,A -85,B 0,C 180,E1 -5287.951,E2 -5287.951} C_VEL
LIN {X 0,Y 515.375,Z 487.63,A -85,B 0,C 180,E1 -5288.292,E2 -5288.292} C_VEL
LIN {X 0,Y 514.15,Z 640.569,A -85,B 0,C 180,E1 -5290.498,E2 -5290.498} C_VEL
LIN {X 0,Y 513.849,Z 655.703,A -85,B 0,C 180,E1 -5290.865,E2 -5290.865} C_VEL
LIN {X 0,Y 513.445,Z 670.716,A -85,B 0,C 180,E1 -5291.393,E2 -5291.393} C_VEL
LIN {X 0,Y 512.904,Z 684.74,A -85,B 0,C 180,E1 -5292.045,E2 -5292.045} C_VEL
LIN {X 0,Y 512.369,Z 698.437,A -85,B 0,C 180,E1 -5292.849,E2 -5292.849} C_VEL
LIN {X 0,Y 511.836,Z 711.165,A -85,B 0,C 180,E1 -5293.766,E2 -5293.766} C_VEL
LIN {X 0,Y 511.235,Z 723.762,A -85,B 0,C 180,E1 -5294.86,E2 -5294.86} C_VEL
LIN {X 0,Y 510.716,Z 735.306,A -85,B 0,C 180,E1 -5296.067,E2 -5296.067} C_VEL
LIN {X 0,Y 510.288,Z 745.04,A -85,B 0,C 180,E1 -5297.271,E2 -5297.271} C_VEL
LIN {X 0,Y 509.977,Z 754.606,A -85,B 0,C 180,E1 -5298.683,E2 -5298.683} C_VEL
LIN {X 0,Y 509.641,Z 762.503,A -85,B 0,C 180,E1 -5300.075,E2 -5300.075} C_VEL
LIN {X 0,Y 509.432,Z 769.906,A -85,B 0,C 180,E1 -5301.672,E2 -5301.672} C_VEL
LIN {X 0,Y 509.256,Z 775.91,A -85,B 0,C 180,E1 -5303.305,E2 -5303.305} C_VEL
LIN {X 0,Y 509.282,Z 779.256,A -85,B 0,C 180,E1 -5304.458,E2 -5304.458} C_VEL
LIN {X 0,Y 509.2,Z 782.795,A -85,B 0,C 180,E1 -5306.044,E2 -5306.044} C_VEL
LIN {X 0,Y 509.158,Z 785.137,A -85,B 0,C 180,E1 -5307.628,E2 -5307.628} C_VEL
LIN {X 0,Y 509.07,Z 786.332,A -85,B 0,C 180,E1 -5309.21,E2 -5309.21} C_VEL
LIN {X 0,Y 509.071,Z 786.351,A -85,B 0,C 180,E1 -5310.792,E2 -5310.792} C_VEL
LIN {X 0,Y 509.159,Z 785.228,A -85,B 0,C 180,E1 -5312.374,E2 -5312.374} C_VEL
LIN {X 0,Y 509.201,Z 782.958,A -85,B 0,C 180,E1 -5313.958,E2 -5313.958} C_VEL
LIN {X 0,Y 509.277,Z 779.487,A -85,B 0,C 180,E1 -5315.545,E2 -5315.545} C_VEL
LIN {X 0,Y 509.32,Z 774.736,A -85,B 0,C 180,E1 -5317.135,E2 -5317.135} C_VEL
LIN {X 0,Y 509.481,Z 768.584,A -85,B 0,C 180,E1 -5318.729,E2 -5318.729} C_VEL
LIN {X 0,Y 509.748,Z 760.845,A -85,B 0,C 180,E1 -5320.326,E2 -5320.326} C_VEL
LIN {X 0,Y 510.012,Z 752.264,A -85,B 0,C 180,E1 -5321.779,E2 -5321.779} C_VEL
LIN {X 0,Y 510.406,Z 742.658,A -85,B 0,C 180,E1 -5323.133,E2 -5323.133} C_VEL
LIN {X 0,Y 510.855,Z 732.523,A -85,B 0,C 180,E1 -5324.339,E2 -5324.339} C_VEL
LIN {X 0,Y 511.367,Z 721.211,A -85,B 0,C 180,E1 -5325.472,E2 -5325.472} C_VEL
LIN {X 0,Y 511.945,Z 708.289,A -85,B 0,C 180,E1 -5326.551,E2 -5326.551} C_VEL
LIN {X 0,Y 512.569,Z 695.119,A -85,B 0,C 180,E1 -5327.455,E2 -5327.455} C_VEL
LIN {X 0,Y 513.05,Z 681.578,A -85,B 0,C 180,E1 -5328.211,E2 -5328.211} C_VEL
LIN {X 0,Y 513.542,Z 666.576,A -85,B 0,C 180,E1 -5328.865,E2 -5328.865} C_VEL
LIN {X 0,Y 513.939,Z 651.719,A -85,B 0,C 180,E1 -5329.342,E2 -5329.342} C_VEL
LIN {X 0,Y 514.229,Z 636.493,A -85,B 0,C 180,E1 -5329.668,E2 -5329.668} C_VEL
LIN {X 0,Y 515.374,Z 487.682,A -85,B 0,C 180,E1 -5331.797,E2 -5331.797} C_VEL
LIN {X 0,Y 513.037,Z 473.24,A -85,B 0,C 180,E1 -5332.12,E2 -5332.12} C_VEL
LIN {X 0,Y 513.044,Z 468.534,A -85,B 0,C 180,E1 -5332.555,E2 -5332.555} C_VEL
LIN {X 0,Y 513.914,Z 438.023,A -85,B 0,C 180,E1 -5335.639,E2 -5335.639} C_VEL
LIN {X 0,Y 514.811,Z 408.685,A -85,B 0,C 180,E1 -5338.689,E2 -5338.689} C_VEL
LIN {X 0,Y 515.439,Z 387.566,A -85,B 0,C 180,E1 -5340.916,E2 -5340.916} C_VEL
LIN {X 0,Y 510.774,Z 371.107,A -85,B 0,C 180,E1 -5342.93,E2 -5342.93} C_VEL
LIN {X 0,Y 509.823,Z 367.754,A -85,B 0,C 180,E1 -5343.399,E2 -5343.399} C_VEL
LIN {X 0,Y 509.752,Z 367.61,A -85,B 0,C 180,E1 -5346.36,E2 -5346.36} C_VEL
LIN {X 0,Y 509.808,Z 367.603,A -85,B 0,C 180,E1 -5349.357,E2 -5349.357} C_VEL
LIN {X 0,Y 509.786,Z 367.6,A -85,B 0,C 180,E1 -5352.496,E2 -5352.496} C_VEL
LIN {X 0,Y 509.838,Z 367.596,A -85,B 0,C 180,E1 -5355.33,E2 -5355.33} C_VEL
LIN {X 0,Y 509.788,Z 367.607,A -85,B 0,C 180,E1 -5358.568,E2 -5358.568} C_VEL
LIN {X 0,Y 509.81,Z 367.605,A -85,B 0,C 180,E1 -5361.658,E2 -5361.658} C_VEL
LIN {X 0,Y 509.81,Z 367.599,A -85,B 0,C 180,E1 -5364.62,E2 -5364.62} C_VEL
LIN {X 0,Y 509.835,Z 367.603,A -85,B 0,C 180,E1 -5367.479,E2 -5367.479} C_VEL
LIN {X 0,Y 509.832,Z 367.6,A -85,B 0,C 180,E1 -5370.28,E2 -5370.28} C_VEL
LIN {X 0,Y 509.818,Z 367.607,A -85,B 0,C 180,E1 -5372.94,E2 -5372.94} C_VEL
LIN {X 0,Y 509.823,Z 367.606,A -85,B 0,C 180,E1 -5375.572,E2 -5375.572} C_VEL
LIN {X 0,Y 509.941,Z 367.781,A -85,B 0,C 180,E1 -5379.042,E2 -5379.042} C_VEL
LIN {X 0,Y 511.355,Z 375.665,A -85,B 0,C 180,E1 -5380.531,E2 -5380.531} C_VEL
LIN {X 0,Y 511.37,Z 379.367,A -85,B 0,C 180,E1 -5381.142,E2 -5381.142} C_VEL
LIN {X 0,Y 513.799,Z 390.528,A -85,B 0,C 180,E1 -5381.434,E2 -5381.434} C_VEL
LIN {X 0,Y 512.774,Z 517.122,A -85,B 0,C 180,E1 -5383.373,E2 -5383.373} C_VEL
LIN {X 0,Y 512.585,Z 530.956,A -85,B 0,C 180,E1 -5383.732,E2 -5383.732} C_VEL
LIN {X 0,Y 512.321,Z 545.436,A -85,B 0,C 180,E1 -5384.28,E2 -5384.28} C_VEL
LIN {X 0,Y 512.005,Z 559.285,A -85,B 0,C 180,E1 -5384.984,E2 -5384.984} C_VEL
LIN {X 0,Y 511.616,Z 571.698,A -85,B 0,C 180,E1 -5385.786,E2 -5385.786} C_VEL
LIN {X 0,Y 511.279,Z 583.033,A -85,B 0,C 180,E1 -5386.688,E2 -5386.688} C_VEL
LIN {X 0,Y 510.906,Z 593.333,A -85,B 0,C 180,E1 -5387.677,E2 -5387.677} C_VEL
LIN {X 0,Y 510.528,Z 603.787,A -85,B 0,C 180,E1 -5388.888,E2 -5388.888} C_VEL
LIN {X 0,Y 510.226,Z 612.291,A -85,B 0,C 180,E1 -5390.085,E2 -5390.085} C_VEL
LIN {X 0,Y 509.982,Z 620.388,A -85,B 0,C 180,E1 -5391.481,E2 -5391.481} C_VEL
LIN {X 0,Y 509.812,Z 626.896,A -85,B 0,C 180,E1 -5392.873,E2 -5392.873} C_VEL
LIN {X 0,Y 509.73,Z 631.403,A -85,B 0,C 180,E1 -5394.064,E2 -5394.064} C_VEL
LIN {X 0,Y 509.561,Z 634.964,A -85,B 0,C 180,E1 -5395.253,E2 -5395.253} C_VEL
LIN {X 0,Y 509.506,Z 638.456,A -85,B 0,C 180,E1 -5396.837,E2 -5396.837} C_VEL
LIN {X 0,Y 509.428,Z 640.576,A -85,B 0,C 180,E1 -5398.419,E2 -5398.419} C_VEL
LIN {X 0,Y 509.459,Z 641.363,A -85,B 0,C 180,E1 -5400,E2 -5400} C_VEL
LIN {X 0,Y 509.428,Z 640.841,A -85,B 0,C 180,E1 -5401.581,E2 -5401.581} C_VEL
LIN {X 0,Y 509.554,Z 638.967,A -85,B 0,C 180,E1 -5403.163,E2 -5403.163} C_VEL
LIN {X 0,Y 509.617,Z 635.736,A -85,B 0,C 180,E1 -5404.746,E2 -5404.746} C_VEL
LIN {X 0,Y 509.859,Z 631.006,A -85,B 0,C 180,E1 -5406.331,E2 -5406.331} C_VEL
LIN {X 0,Y 509.9,Z 626.423,A -85,B 0,C 180,E1 -5407.524,E2 -5407.524} C_VEL
LIN {X 0,Y 510.167,Z 619.713,A -85,B 0,C 180,E1 -5408.915,E2 -5408.915} C_VEL
LIN {X 0,Y 510.438,Z 611.349,A -85,B 0,C 180,E1 -5410.311,E2 -5410.311} C_VEL
LIN {X 0,Y 510.845,Z 602.534,A -85,B 0,C 180,E1 -5411.507,E2 -5411.507} C_VEL
LIN {X 0,Y 511.176,Z 593.467,A -85,B 0,C 180,E1 -5412.535,E2 -5412.535} C_VEL
LIN {X 0,Y 511.534,Z 582.07,A -85,B 0,C 180,E1 -5413.608,E2 -5413.608} C_VEL
LIN {X 0,Y 511.836,Z 570.285,A -85,B 0,C 180,E1 -5414.512,E2 -5414.512} C_VEL
LIN {X 0,Y 512.198,Z 557.145,A -85,B 0,C 180,E1 -5415.315,E2 -5415.315} C_VEL
LIN {X 0,Y 512.455,Z 544.49,A -85,B 0,C 180,E1 -5415.919,E2 -5415.919} C_VEL
LIN {X 0,Y 512.675,Z 530.417,A -85,B 0,C 180,E1 -5416.417,E2 -5416.417} C_VEL
LIN {X 0,Y 512.814,Z 516.353,A -85,B 0,C 180,E1 -5416.752,E2 -5416.752} C_VEL
LIN {X 0,Y 514.179,Z 403.909,A -85,B 0,C 180,E1 -5418.58,E2 -5418.58} C_VEL
LIN {X 0,Y 514.334,Z 390.568,A -85,B 0,C 180,E1 -5418.81,E2 -5418.81} C_VEL
LIN {X 0,Y 512.487,Z 383.745,A -85,B 0,C 180,E1 -5419.043,E2 -5419.043} C_VEL
LIN {X 0,Y 512.518,Z 379.309,A -85,B 0,C 180,E1 -5419.84,E2 -5419.84} C_VEL
LIN {X 0,Y 510.42,Z 369.976,A -85,B 0,C 180,E1 -5421.824,E2 -5421.824} C_VEL
LIN {X 0,Y 509.847,Z 367.685,A -85,B 0,C 180,E1 -5422.343,E2 -5422.343} C_VEL
LIN {X 0,Y 509.881,Z 367.598,A -85,B 0,C 180,E1 -5425.296,E2 -5425.296} C_VEL
LIN {X 0,Y 509.901,Z 367.594,A -85,B 0,C 180,E1 -5428.1,E2 -5428.1} C_VEL
LIN {X 0,Y 509.85,Z 367.601,A -85,B 0,C 180,E1 -5431.279,E2 -5431.279} C_VEL
LIN {X 0,Y 509.86,Z 367.602,A -85,B 0,C 180,E1 -5434.202,E2 -5434.202} C_VEL
LIN {X 0,Y 509.812,Z 367.604,A -85,B 0,C 180,E1 -5437.341,E2 -5437.341} C_VEL
LIN {X 0,Y 509.842,Z 367.605,A -85,B 0,C 180,E1 -5440.382,E2 -5440.382} C_VEL
LIN {X 0,Y 509.804,Z 367.605,A -85,B 0,C 180,E1 -5443.059,E2 -5443.059} C_VEL
LIN {X 0,Y 509.825,Z 367.605,A -85,B 0,C 180,E1 -5445.793,E2 -5445.793} C_VEL
LIN {X 0,Y 509.833,Z 367.605,A -85,B 0,C 180,E1 -5448.571,E2 -5448.571} C_VEL
LIN {X 0,Y 509.817,Z 367.608,A -85,B 0,C 180,E1 -5451.791,E2 -5451.791} C_VEL
LIN {X 0,Y 509.809,Z 367.608,A -85,B 0,C 180,E1 -5454.619,E2 -5454.619} C_VEL
LIN {X 0,Y 509.883,Z 367.811,A -85,B 0,C 180,E1 -5457.715,E2 -5457.715} C_VEL
LIN {X 0,Y 512.851,Z 378.156,A -85,B 0,C 180,E1 -5459.076,E2 -5459.076} C_VEL
LIN {X 0,Y 514.977,Z 386.884,A -85,B 0,C 180,E1 -5460.123,E2 -5460.123} C_VEL
LIN {X 0,Y 513.975,Z 415.101,A -85,B 0,C 180,E1 -5462.934,E2 -5462.934} C_VEL
LIN {X 0,Y 513.04,Z 446.399,A -85,B 0,C 180,E1 -5465.949,E2 -5465.949} C_VEL
LIN {X 0,Y 512.504,Z 468.338,A -85,B 0,C 180,E1 -5467.995,E2 -5467.995} C_VEL
LIN {X 0,Y 514.86,Z 486.977,A -85,B 0,C 180,E1 -5468.397,E2 -5468.397} C_VEL
LIN {X 0,Y 513.776,Z 615.535,A -85,B 0,C 180,E1 -5470.288,E2 -5470.288} C_VEL
LIN {X 0,Y 513.561,Z 639.863,A -85,B 0,C 180,E1 -5470.669,E2 -5470.669} C_VEL
LIN {X 0,Y 513.181,Z 657.649,A -85,B 0,C 180,E1 -5471.124,E2 -5471.124} C_VEL
LIN {X 0,Y 512.777,Z 672.586,A -85,B 0,C 180,E1 -5471.676,E2 -5471.676} C_VEL
LIN {X 0,Y 512.378,Z 686.125,A -85,B 0,C 180,E1 -5472.332,E2 -5472.332} C_VEL
LIN {X 0,Y 511.835,Z 699.43,A -85,B 0,C 180,E1 -5473.137,E2 -5473.137} C_VEL
LIN {X 0,Y 511.329,Z 713.295,A -85,B 0,C 180,E1 -5474.179,E2 -5474.179} C_VEL
LIN {X 0,Y 510.839,Z 725.132,A -85,B 0,C 180,E1 -5475.254,E2 -5475.254} C_VEL
LIN {X 0,Y 510.365,Z 738.07,A -85,B 0,C 180,E1 -5476.663,E2 -5476.663} C_VEL
LIN {X 0,Y 509.966,Z 749.047,A -85,B 0,C 180,E1 -5478.09,E2 -5478.09} C_VEL
LIN {X 0,Y 509.756,Z 757.91,A -85,B 0,C 180,E1 -5479.473,E2 -5479.473} C_VEL
LIN {X 0,Y 509.51,Z 765.377,A -85,B 0,C 180,E1 -5480.872,E2 -5480.872} C_VEL
LIN {X 0,Y 509.353,Z 772.302,A -85,B 0,C 180,E1 -5482.467,E2 -5482.467} C_VEL
LIN {X 0,Y 509.291,Z 777.713,A -85,B 0,C 180,E1 -5484.058,E2 -5484.058} C_VEL
LIN {X 0,Y 509.159,Z 780.815,A -85,B 0,C 180,E1 -5485.248,E2 -5485.248} C_VEL
LIN {X 0,Y 509.189,Z 783.862,A -85,B 0,C 180,E1 -5486.834,E2 -5486.834} C_VEL
LIN {X 0,Y 509.11,Z 785.666,A -85,B 0,C 180,E1 -5488.417,E2 -5488.417} C_VEL
LIN {X 0,Y 509.062,Z 786.282,A -85,B 0,C 180,E1 -5489.999,E2 -5489.999} C_VEL
LIN {X 0,Y 509.109,Z 785.67,A -85,B 0,C 180,E1 -5491.581,E2 -5491.581} C_VEL
LIN {X 0,Y 509.188,Z 783.875,A -85,B 0,C 180,E1 -5493.164,E2 -5493.164} C_VEL
LIN {X 0,Y 509.158,Z 780.841,A -85,B 0,C 180,E1 -5494.749,E2 -5494.749} C_VEL
LIN {X 0,Y 509.284,Z 777.75,A -85,B 0,C 180,E1 -5495.939,E2 -5495.939} C_VEL
LIN {X 0,Y 509.351,Z 772.383,A -85,B 0,C 180,E1 -5497.531,E2 -5497.531} C_VEL
LIN {X 0,Y 509.515,Z 765.526,A -85,B 0,C 180,E1 -5499.126,E2 -5499.126} C_VEL
LIN {X 0,Y 509.755,Z 758.138,A -85,B 0,C 180,E1 -5500.524,E2 -5500.524} C_VEL
LIN {X 0,Y 509.961,Z 749.24,A -85,B 0,C 180,E1 -5501.929,E2 -5501.929} C_VEL
LIN {X 0,Y 510.362,Z 738.553,A -85,B 0,C 180,E1 -5503.334,E2 -5503.334} C_VEL
LIN {X 0,Y 510.803,Z 726.598,A -85,B 0,C 180,E1 -5504.643,E2 -5504.643} C_VEL
LIN {X 0,Y 511.327,Z 713.638,A -85,B 0,C 180,E1 -5505.82,E2 -5505.82} C_VEL
LIN {X 0,Y 511.821,Z 701.234,A -85,B 0,C 180,E1 -5506.758,E2 -5506.758} C_VEL
LIN {X 0,Y 512.354,Z 686.615,A -85,B 0,C 180,E1 -5507.666,E2 -5507.666} C_VEL
LIN {X 0,Y 512.866,Z 672.328,A -85,B 0,C 180,E1 -5508.37,E2 -5508.37} C_VEL
LIN {X 0,Y 513.305,Z 656.999,A -85,B 0,C 180,E1 -5508.949,E2 -5508.949} C_VEL
LIN {X 0,Y 513.667,Z 641.812,A -85,B 0,C 180,E1 -5509.355,E2 -5509.355} C_VEL
LIN {X 0,Y 513.894,Z 620.425,A -85,B 0,C 180,E1 -5509.704,E2 -5509.704} C_VEL
LIN {X 0,Y 515.043,Z 485.984,A -85,B 0,C 180,E1 -5511.67,E2 -5511.67} C_VEL
LIN {X 0,Y 512.782,Z 470.117,A -85,B 0,C 180,E1 -5512.019,E2 -5512.019} C_VEL
LIN {X 0,Y 513.75,Z 438.093,A -85,B 0,C 180,E1 -5515.09,E2 -5515.09} C_VEL
LIN {X 0,Y 514.844,Z 406.04,A -85,B 0,C 180,E1 -5518.205,E2 -5518.205} C_VEL
LIN {X 0,Y 515.468,Z 387.428,A -85,B 0,C 180,E1 -5520.068,E2 -5520.068} C_VEL
LIN {X 0,Y 509.914,Z 367.9,A -85,B 0,C 180,E1 -5522.439,E2 -5522.439} C_VEL
LIN {X 0,Y 509.835,Z 367.603,A -85,B 0,C 180,E1 -5522.767,E2 -5522.767} C_VEL
LIN {X 0,Y 509.785,Z 367.607,A -85,B 0,C 180,E1 -5525.572,E2 -5525.572} C_VEL
LIN {X 0,Y 509.804,Z 367.611,A -85,B 0,C 180,E1 -5528.34,E2 -5528.34} C_VEL
LIN {X 0,Y 509.819,Z 367.602,A -85,B 0,C 180,E1 -5531.427,E2 -5531.427} C_VEL
LIN {X 0,Y 509.827,Z 367.604,A -85,B 0,C 180,E1 -5534.669,E2 -5534.669} C_VEL
LIN {X 0,Y 509.772,Z 367.594,A -85,B 0,C 180,E1 -5537.504,E2 -5537.504} C_VEL
LIN {X 0,Y 509.818,Z 367.606,A -85,B 0,C 180,E1 -5540.645,E2 -5540.645} C_VEL
LIN {X 0,Y 509.752,Z 367.601,A -85,B 0,C 180,E1 -5543.641,E2 -5543.641} C_VEL
LIN {X 0,Y 509.824,Z 367.597,A -85,B 0,C 180,E1 -5546.537,E2 -5546.537} C_VEL
LIN {X 0,Y 509.818,Z 367.6,A -85,B 0,C 180,E1 -5549.332,E2 -5549.332} C_VEL
LIN {X 0,Y 509.816,Z 367.601,A -85,B 0,C 180,E1 -5552.05,E2 -5552.05} C_VEL
LIN {X 0,Y 509.789,Z 367.603,A -85,B 0,C 180,E1 -5554.699,E2 -5554.699} C_VEL
LIN {X 0,Y 509.808,Z 367.602,A -85,B 0,C 180,E1 -5557.458,E2 -5557.458} C_VEL
LIN {X 0,Y 509.889,Z 367.589,A -85,B 0,C 180,E1 -5559.844,E2 -5559.844} C_VEL
LIN {X 0,Y 509.829,Z 367.605,A -85,B 0,C 180,E1 -5562.346,E2 -5562.346} C_VEL
LIN {X 0,Y 509.867,Z 367.592,A -85,B 0,C 180,E1 -5564.818,E2 -5564.818} C_VEL
LIN {X 0,Y 509.884,Z 367.596,A -85,B 0,C 180,E1 -5568.124,E2 -5568.124} C_VEL
LIN {X 0,Y 509.86,Z 367.592,A -85,B 0,C 180,E1 -5571.279,E2 -5571.279} C_VEL
LIN {X 0,Y 509.879,Z 367.592,A -85,B 0,C 180,E1 -5573.669,E2 -5573.669} C_VEL
LIN {X 0,Y 509.903,Z 367.593,A -85,B 0,C 180,E1 -5576.84,E2 -5576.84} C_VEL
LIN {X 0,Y 509.915,Z 367.594,A -85,B 0,C 180,E1 -5578.421,E2 -5578.421} C_VEL
LIN {X 0,Y 510.044,Z 367.571,A -85,B 0,C 180,E1 -5580.79,E2 -5580.79} C_VEL
LIN {X 0,Y 509.893,Z 367.593,A -85,B 0,C 180,E1 -5583.161,E2 -5583.161} C_VEL
LIN {X 0,Y 509.919,Z 367.589,A -85,B 0,C 180,E1 -5586.33,E2 -5586.33} C_VEL
LIN {X 0,Y 509.866,Z 367.601,A -85,B 0,C 180,E1 -5588.721,E2 -5588.721} C_VEL
LIN {X 0,Y 509.888,Z 367.585,A -85,B 0,C 180,E1 -5591.932,E2 -5591.932} C_VEL
LIN {X 0,Y 509.879,Z 367.591,A -85,B 0,C 180,E1 -5595.242,E2 -5595.242} C_VEL
LIN {X 0,Y 509.841,Z 367.601,A -85,B 0,C 180,E1 -5598.485,E2 -5598.485} C_VEL
LIN {X 0,Y 509.834,Z 367.598,A -85,B 0,C 180,E1 -5601.002,E2 -5601.002} C_VEL
LIN {X 0,Y 509.802,Z 367.603,A -85,B 0,C 180,E1 -5603.565,E2 -5603.565} C_VEL
LIN {X 0,Y 509.791,Z 367.604,A -85,B 0,C 180,E1 -5606.355,E2 -5606.355} C_VEL
LIN {X 0,Y 509.819,Z 367.603,A -85,B 0,C 180,E1 -5608.848,E2 -5608.848} C_VEL
LIN {X 0,Y 509.783,Z 367.606,A -85,B 0,C 180,E1 -5611.593,E2 -5611.593} C_VEL
LIN {X 0,Y 509.823,Z 367.605,A -85,B 0,C 180,E1 -5614.416,E2 -5614.416} C_VEL
LIN {X 0,Y 509.779,Z 367.595,A -85,B 0,C 180,E1 -5617.344,E2 -5617.344} C_VEL
LIN {X 0,Y 509.8,Z 367.607,A -85,B 0,C 180,E1 -5620.386,E2 -5620.386} C_VEL
LIN {X 0,Y 509.78,Z 367.605,A -85,B 0,C 180,E1 -5623.576,E2 -5623.576} C_VEL
LIN {X 0,Y 509.781,Z 367.605,A -85,B 0,C 180,E1 -5626.426,E2 -5626.426} C_VEL
LIN {X 0,Y 509.802,Z 367.6,A -85,B 0,C 180,E1 -5629.617,E2 -5629.617} C_VEL
LIN {X 0,Y 509.773,Z 367.607,A -85,B 0,C 180,E1 -5632.658,E2 -5632.658} C_VEL
LIN {X 0,Y 509.759,Z 367.612,A -85,B 0,C 180,E1 -5633.751,E2 -5633.751} C_VEL
LIN {X 0,Y 509.084,Z 367.698,A -85,B 0,C 180,E1 -5634.192,E2 -5634.192} C_VEL
LIN {X 0,Y 506.25,Z 368.042,A -85,B 0,C 180,E1 -5634.881,E2 -5634.881} C_VEL
LIN {X 0,Y 503.427,Z 368.377,A -85,B 0,C 180,E1 -5635.578,E2 -5635.578} C_VEL
LIN {X 0,Y 502.783,Z 368.453,A -85,B 0,C 180,E1 -5636.027,E2 -5636.027} C_VEL
LIN {X 0,Y 502.841,Z 368.757,A -85,B 0,C 180,E1 -5636.394,E2 -5636.394} C_VEL
LIN {X 0,Y 508.068,Z 386.994,A -85,B 0,C 180,E1 -5638.695,E2 -5638.695} C_VEL
LIN {X 0,Y 508.806,Z 390.102,A -85,B 0,C 180,E1 -5639.072,E2 -5639.072} C_VEL
LIN {X 0,Y 507.82,Z 419.799,A -85,B 0,C 180,E1 -5642.221,E2 -5642.221} C_VEL
LIN {X 0,Y 506.834,Z 449.441,A -85,B 0,C 180,E1 -5645.311,E2 -5645.311} C_VEL
LIN {X 0,Y 506.213,Z 472.426,A -85,B 0,C 180,E1 -5647.621,E2 -5647.621} C_VEL
LIN {X 0,Y 507.225,Z 478.736,A -85,B 0,C 180,E1 -5647.794,E2 -5647.794} C_VEL
LIN {X 0,Y 508.733,Z 487.769,A -85,B 0,C 180,E1 -5647.998,E2 -5647.998} C_VEL
LIN {X 0,Y 507.481,Z 640.581,A -85,B 0,C 180,E1 -5650.234,E2 -5650.234} C_VEL
LIN {X 0,Y 507.139,Z 656.483,A -85,B 0,C 180,E1 -5650.628,E2 -5650.628} C_VEL
LIN {X 0,Y 506.69,Z 670.664,A -85,B 0,C 180,E1 -5651.136,E2 -5651.136} C_VEL
LIN {X 0,Y 506.124,Z 684.699,A -85,B 0,C 180,E1 -5651.796,E2 -5651.796} C_VEL
LIN {X 0,Y 505.558,Z 698.404,A -85,B 0,C 180,E1 -5652.611,E2 -5652.611} C_VEL
LIN {X 0,Y 505.004,Z 711.007,A -85,B 0,C 180,E1 -5653.529,E2 -5653.529} C_VEL
LIN {X 0,Y 504.357,Z 723.739,A -85,B 0,C 180,E1 -5654.649,E2 -5654.649} C_VEL
LIN {X 0,Y 503.749,Z 735.287,A -85,B 0,C 180,E1 -5655.87,E2 -5655.87} C_VEL
LIN {X 0,Y 503.305,Z 745.023,A -85,B 0,C 180,E1 -5657.092,E2 -5657.092} C_VEL
LIN {X 0,Y 502.927,Z 754.717,A -85,B 0,C 180,E1 -5658.544,E2 -5658.544} C_VEL
LIN {X 0,Y 502.603,Z 762.488,A -85,B 0,C 180,E1 -5659.935,E2 -5659.935} C_VEL
LIN {X 0,Y 502.374,Z 769.892,A -85,B 0,C 180,E1 -5661.555,E2 -5661.555} C_VEL
LIN {X 0,Y 502.189,Z 775.896,A -85,B 0,C 180,E1 -5663.21,E2 -5663.21} C_VEL
LIN {X 0,Y 502.195,Z 779.243,A -85,B 0,C 180,E1 -5664.38,E2 -5664.38} C_VEL
LIN {X 0,Y 502.096,Z 782.782,A -85,B 0,C 180,E1 -5665.988,E2 -5665.988} C_VEL
LIN {X 0,Y 502.062,Z 785.123,A -85,B 0,C 180,E1 -5667.594,E2 -5667.594} C_VEL
LIN {X 0,Y 501.987,Z 786.319,A -85,B 0,C 180,E1 -5669.199,E2 -5669.199} C_VEL
LIN {X 0,Y 501.988,Z 786.337,A -85,B 0,C 180,E1 -5670.803,E2 -5670.803} C_VEL
LIN {X 0,Y 502.063,Z 785.213,A -85,B 0,C 180,E1 -5672.408,E2 -5672.408} C_VEL
LIN {X 0,Y 502.096,Z 782.942,A -85,B 0,C 180,E1 -5674.014,E2 -5674.014} C_VEL
LIN {X 0,Y 502.186,Z 779.47,A -85,B 0,C 180,E1 -5675.623,E2 -5675.623} C_VEL
LIN {X 0,Y 502.246,Z 774.718,A -85,B 0,C 180,E1 -5677.236,E2 -5677.236} C_VEL
LIN {X 0,Y 502.413,Z 768.564,A -85,B 0,C 180,E1 -5678.853,E2 -5678.853} C_VEL
LIN {X 0,Y 502.74,Z 760.824,A -85,B 0,C 180,E1 -5680.472,E2 -5680.472} C_VEL
LIN {X 0,Y 502.982,Z 752.799,A -85,B 0,C 180,E1 -5681.859,E2 -5681.859} C_VEL
LIN {X 0,Y 503.343,Z 744.185,A -85,B 0,C 180,E1 -5683.115,E2 -5683.115} C_VEL
LIN {X 0,Y 503.829,Z 734.281,A -85,B 0,C 180,E1 -5684.336,E2 -5684.336} C_VEL
LIN {X 0,Y 504.384,Z 723.041,A -85,B 0,C 180,E1 -5685.509,E2 -5685.509} C_VEL
LIN {X 0,Y 504.977,Z 710.801,A -85,B 0,C 180,E1 -5686.578,E2 -5686.578} C_VEL
LIN {X 0,Y 505.624,Z 698.161,A -85,B 0,C 180,E1 -5687.493,E2 -5687.493} C_VEL
LIN {X 0,Y 506.148,Z 684.387,A -85,B 0,C 180,E1 -5688.311,E2 -5688.311} C_VEL
LIN {X 0,Y 506.703,Z 669.623,A -85,B 0,C 180,E1 -5688.997,E2 -5688.997} C_VEL
LIN {X 0,Y 507.107,Z 654.555,A -85,B 0,C 180,E1 -5689.522,E2 -5689.522} C_VEL
LIN {X 0,Y 507.438,Z 639.393,A -85,B 0,C 180,E1 -5689.882,E2 -5689.882} C_VEL
LIN {X 0,Y 508.801,Z 489.286,A -85,B 0,C 180,E1 -5692.066,E2 -5692.066} C_VEL
LIN {X 0,Y 506.28,Z 473.034,A -85,B 0,C 180,E1 -5692.434,E2 -5692.434} C_VEL
LIN {X 0,Y 506.248,Z 469.434,A -85,B 0,C 180,E1 -5692.767,E2 -5692.767} C_VEL
LIN {X 0,Y 507.046,Z 441.693,A -85,B 0,C 180,E1 -5695.577,E2 -5695.577} C_VEL
LIN {X 0,Y 507.883,Z 415.819,A -85,B 0,C 180,E1 -5698.292,E2 -5698.292} C_VEL
LIN {X 0,Y 508.791,Z 391.611,A -85,B 0,C 180,E1 -5700.86,E2 -5700.86} C_VEL
LIN {X 0,Y 508.757,Z 389.624,A -85,B 0,C 180,E1 -5701.077,E2 -5701.077} C_VEL
LIN {X 0,Y 503.905,Z 372.611,A -85,B 0,C 180,E1 -5703.193,E2 -5703.193} C_VEL
LIN {X 0,Y 502.763,Z 368.658,A -85,B 0,C 180,E1 -5703.732,E2 -5703.732} C_VEL
LIN {X 0,Y 502.698,Z 368.488,A -85,B 0,C 180,E1 -5706.954,E2 -5706.954} C_VEL
LIN {X 0,Y 502.734,Z 368.487,A -85,B 0,C 180,E1 -5709.747,E2 -5709.747} C_VEL
LIN {X 0,Y 502.749,Z 368.475,A -85,B 0,C 180,E1 -5712.192,E2 -5712.192} C_VEL
LIN {X 0,Y 502.781,Z 368.474,A -85,B 0,C 180,E1 -5715.472,E2 -5715.472} C_VEL
LIN {X 0,Y 502.754,Z 368.482,A -85,B 0,C 180,E1 -5718.927,E2 -5718.927} C_VEL
LIN {X 0,Y 502.757,Z 368.481,A -85,B 0,C 180,E1 -5722.043,E2 -5722.043} C_VEL
LIN {X 0,Y 502.784,Z 368.47,A -85,B 0,C 180,E1 -5725.033,E2 -5725.033} C_VEL
LIN {X 0,Y 502.76,Z 368.481,A -85,B 0,C 180,E1 -5727.914,E2 -5727.914} C_VEL
LIN {X 0,Y 502.793,Z 368.48,A -85,B 0,C 180,E1 -5730.71,E2 -5730.71} C_VEL
LIN {X 0,Y 502.774,Z 368.483,A -85,B 0,C 180,E1 -5733.461,E2 -5733.461} C_VEL
LIN {X 0,Y 502.76,Z 368.483,A -85,B 0,C 180,E1 -5736.085,E2 -5736.085} C_VEL
LIN {X 0,Y 502.854,Z 368.603,A -85,B 0,C 180,E1 -5738.807,E2 -5738.807} C_VEL
LIN {X 0,Y 504.458,Z 377.299,A -85,B 0,C 180,E1 -5740.466,E2 -5740.466} C_VEL
LIN {X 0,Y 504.506,Z 379.955,A -85,B 0,C 180,E1 -5740.878,E2 -5740.878} C_VEL
LIN {X 0,Y 507.106,Z 391.416,A -85,B 0,C 180,E1 -5741.185,E2 -5741.185} C_VEL
LIN {X 0,Y 505.941,Z 518.183,A -85,B 0,C 180,E1 -5743.168,E2 -5743.168} C_VEL
LIN {X 0,Y 505.757,Z 532.288,A -85,B 0,C 180,E1 -5743.546,E2 -5743.546} C_VEL
LIN {X 0,Y 505.488,Z 546.88,A -85,B 0,C 180,E1 -5744.114,E2 -5744.114} C_VEL
LIN {X 0,Y 505.183,Z 559.712,A -85,B 0,C 180,E1 -5744.776,E2 -5744.776} C_VEL
LIN {X 0,Y 504.825,Z 570.78,A -85,B 0,C 180,E1 -5745.487,E2 -5745.487} C_VEL
LIN {X 0,Y 504.44,Z 582.442,A -85,B 0,C 180,E1 -5746.402,E2 -5746.402} C_VEL
LIN {X 0,Y 504.043,Z 593.263,A -85,B 0,C 180,E1 -5747.431,E2 -5747.431} C_VEL
LIN {X 0,Y 503.751,Z 602.865,A -85,B 0,C 180,E1 -5748.533,E2 -5748.533} C_VEL
LIN {X 0,Y 503.355,Z 611.705,A -85,B 0,C 180,E1 -5749.746,E2 -5749.746} C_VEL
LIN {X 0,Y 503.092,Z 619.035,A -85,B 0,C 180,E1 -5750.958,E2 -5750.958} C_VEL
LIN {X 0,Y 502.864,Z 626.037,A -85,B 0,C 180,E1 -5752.37,E2 -5752.37} C_VEL
LIN {X 0,Y 502.772,Z 630.873,A -85,B 0,C 180,E1 -5753.579,E2 -5753.579} C_VEL
LIN {X 0,Y 502.549,Z 635.9,A -85,B 0,C 180,E1 -5755.187,E2 -5755.187} C_VEL
LIN {X 0,Y 502.483,Z 639.431,A -85,B 0,C 180,E1 -5756.793,E2 -5756.793} C_VEL
LIN {X 0,Y 502.412,Z 641.58,A -85,B 0,C 180,E1 -5758.397,E2 -5758.397} C_VEL
LIN {X 0,Y 502.449,Z 642.387,A -85,B 0,C 180,E1 -5760,E2 -5760} C_VEL
LIN {X 0,Y 502.412,Z 641.879,A -85,B 0,C 180,E1 -5761.603,E2 -5761.603} C_VEL
LIN {X 0,Y 502.54,Z 640.011,A -85,B 0,C 180,E1 -5763.207,E2 -5763.207} C_VEL
LIN {X 0,Y 502.614,Z 636.777,A -85,B 0,C 180,E1 -5764.813,E2 -5764.813} C_VEL
LIN {X 0,Y 502.882,Z 632.035,A -85,B 0,C 180,E1 -5766.419,E2 -5766.419} C_VEL
LIN {X 0,Y 502.933,Z 627.435,A -85,B 0,C 180,E1 -5767.629,E2 -5767.629} C_VEL
LIN {X 0,Y 503.223,Z 620.711,A -85,B 0,C 180,E1 -5769.04,E2 -5769.04} C_VEL
LIN {X 0,Y 503.527,Z 612.329,A -85,B 0,C 180,E1 -5770.454,E2 -5770.454} C_VEL
LIN {X 0,Y 503.958,Z 603.493,A -85,B 0,C 180,E1 -5771.666,E2 -5771.666} C_VEL
LIN {X 0,Y 504.317,Z 594.397,A -85,B 0,C 180,E1 -5772.707,E2 -5772.707} C_VEL
LIN {X 0,Y 504.695,Z 582.938,A -85,B 0,C 180,E1 -5773.796,E2 -5773.796} C_VEL
LIN {X 0,Y 505.009,Z 571.093,A -85,B 0,C 180,E1 -5774.713,E2 -5774.713} C_VEL
LIN {X 0,Y 505.389,Z 557.828,A -85,B 0,C 180,E1 -5775.527,E2 -5775.527} C_VEL
LIN {X 0,Y 505.755,Z 543.856,A -85,B 0,C 180,E1 -5776.185,E2 -5776.185} C_VEL
LIN {X 0,Y 505.911,Z 529.752,A -85,B 0,C 180,E1 -5776.675,E2 -5776.675} C_VEL
LIN {X 0,Y 506.073,Z 515.179,A -85,B 0,C 180,E1 -5777.008,E2 -5777.008} C_VEL
LIN {X 0,Y 507.512,Z 410.711,A -85,B 0,C 180,E1 -5778.758,E2 -5778.758} C_VEL
LIN {X 0,Y 507.763,Z 391.914,A -85,B 0,C 180,E1 -5779.093,E2 -5779.093} C_VEL
LIN {X 0,Y 505.839,Z 384.775,A -85,B 0,C 180,E1 -5779.349,E2 -5779.349} C_VEL
LIN {X 0,Y 505.691,Z 380.602,A -85,B 0,C 180,E1 -5780.119,E2 -5780.119} C_VEL
LIN {X 0,Y 503.493,Z 371.318,A -85,B 0,C 180,E1 -5782.14,E2 -5782.14} C_VEL
LIN {X 0,Y 502.795,Z 368.517,A -85,B 0,C 180,E1 -5782.822,E2 -5782.822} C_VEL
LIN {X 0,Y 502.844,Z 368.474,A -85,B 0,C 180,E1 -5785.675,E2 -5785.675} C_VEL
LIN {X 0,Y 502.845,Z 368.475,A -85,B 0,C 180,E1 -5788.372,E2 -5788.372} C_VEL
LIN {X 0,Y 502.797,Z 368.479,A -85,B 0,C 180,E1 -5791.498,E2 -5791.498} C_VEL
LIN {X 0,Y 502.808,Z 368.478,A -85,B 0,C 180,E1 -5793.994,E2 -5793.994} C_VEL
LIN {X 0,Y 502.769,Z 368.482,A -85,B 0,C 180,E1 -5797.175,E2 -5797.175} C_VEL
LIN {X 0,Y 502.791,Z 368.482,A -85,B 0,C 180,E1 -5800.015,E2 -5800.015} C_VEL
LIN {X 0,Y 502.807,Z 368.481,A -85,B 0,C 180,E1 -5802.199,E2 -5802.199} C_VEL
LIN {X 0,Y 502.789,Z 368.479,A -85,B 0,C 180,E1 -5805.47,E2 -5805.47} C_VEL
LIN {X 0,Y 502.774,Z 368.482,A -85,B 0,C 180,E1 -5808.929,E2 -5808.929} C_VEL
LIN {X 0,Y 502.762,Z 368.488,A -85,B 0,C 180,E1 -5812.042,E2 -5812.042} C_VEL
LIN {X 0,Y 502.783,Z 368.483,A -85,B 0,C 180,E1 -5815.032,E2 -5815.032} C_VEL
LIN {X 0,Y 502.838,Z 368.708,A -85,B 0,C 180,E1 -5817.326,E2 -5817.326} C_VEL
LIN {X 0,Y 506.216,Z 380.298,A -85,B 0,C 180,E1 -5818.897,E2 -5818.897} C_VEL
LIN {X 0,Y 508.326,Z 388.922,A -85,B 0,C 180,E1 -5819.958,E2 -5819.958} C_VEL
LIN {X 0,Y 507.172,Z 416.696,A -85,B 0,C 180,E1 -5822.787,E2 -5822.787} C_VEL
LIN {X 0,Y 506.139,Z 447.571,A -85,B 0,C 180,E1 -5825.818,E2 -5825.818} C_VEL
LIN {X 0,Y 505.6,Z 467.456,A -85,B 0,C 180,E1 -5827.698,E2 -5827.698} C_VEL
LIN {X 0,Y 508.171,Z 487.389,A -85,B 0,C 180,E1 -5828.143,E2 -5828.143} C_VEL
LIN {X 0,Y 507.348,Z 579.424,A -85,B 0,C 180,E1 -5829.525,E2 -5829.525} C_VEL
LIN {X 0,Y 506.773,Z 641.93,A -85,B 0,C 180,E1 -5830.453,E2 -5830.453} C_VEL
LIN {X 0,Y 506.478,Z 657.334,A -85,B 0,C 180,E1 -5830.851,E2 -5830.851} C_VEL
LIN {X 0,Y 506.094,Z 671.513,A -85,B 0,C 180,E1 -5831.373,E2 -5831.373} C_VEL
LIN {X 0,Y 505.599,Z 686.19,A -85,B 0,C 180,E1 -5832.088,E2 -5832.088} C_VEL
LIN {X 0,Y 505.027,Z 699.477,A -85,B 0,C 180,E1 -5832.903,E2 -5832.903} C_VEL
LIN {X 0,Y 504.463,Z 712.9,A -85,B 0,C 180,E1 -5833.92,E2 -5833.92} C_VEL
LIN {X 0,Y 503.923,Z 725.17,A -85,B 0,C 180,E1 -5835.047,E2 -5835.047} C_VEL
LIN {X 0,Y 503.466,Z 736.29,A -85,B 0,C 180,E1 -5836.271,E2 -5836.271} C_VEL
LIN {X 0,Y 503.074,Z 745.646,A -85,B 0,C 180,E1 -5837.493,E2 -5837.493} C_VEL
LIN {X 0,Y 502.749,Z 754.815,A -85,B 0,C 180,E1 -5838.917,E2 -5838.917} C_VEL
LIN {X 0,Y 502.455,Z 762.406,A -85,B 0,C 180,E1 -5840.336,E2 -5840.336} C_VEL
LIN {X 0,Y 502.373,Z 769.598,A -85,B 0,C 180,E1 -5841.957,E2 -5841.957} C_VEL
LIN {X 0,Y 502.254,Z 775.401,A -85,B 0,C 180,E1 -5843.571,E2 -5843.571} C_VEL
LIN {X 0,Y 502.137,Z 779.771,A -85,B 0,C 180,E1 -5845.182,E2 -5845.182} C_VEL
LIN {X 0,Y 502.148,Z 782.847,A -85,B 0,C 180,E1 -5846.79,E2 -5846.79} C_VEL
LIN {X 0,Y 502.077,Z 784.677,A -85,B 0,C 180,E1 -5848.395,E2 -5848.395} C_VEL
LIN {X 0,Y 502.03,Z 785.308,A -85,B 0,C 180,E1 -5849.999,E2 -5849.999} C_VEL
LIN {X 0,Y 502.074,Z 784.706,A -85,B 0,C 180,E1 -5851.603,E2 -5851.603} C_VEL
LIN {X 0,Y 502.14,Z 782.91,A -85,B 0,C 180,E1 -5853.208,E2 -5853.208} C_VEL
LIN {X 0,Y 502.136,Z 779.875,A -85,B 0,C 180,E1 -5854.816,E2 -5854.816} C_VEL
LIN {X 0,Y 502.212,Z 775.553,A -85,B 0,C 180,E1 -5856.427,E2 -5856.427} C_VEL
LIN {X 0,Y 502.339,Z 769.832,A -85,B 0,C 180,E1 -5858.041,E2 -5858.041} C_VEL
LIN {X 0,Y 502.482,Z 762.539,A -85,B 0,C 180,E1 -5859.661,E2 -5859.661} C_VEL
LIN {X 0,Y 502.793,Z 753.6,A -85,B 0,C 180,E1 -5861.284,E2 -5861.284} C_VEL
LIN {X 0,Y 503.042,Z 745.674,A -85,B 0,C 180,E1 -5862.505,E2 -5862.505} C_VEL
LIN {X 0,Y 503.497,Z 734.564,A -85,B 0,C 180,E1 -5863.931,E2 -5863.931} C_VEL
LIN {X 0,Y 503.971,Z 723.099,A -85,B 0,C 180,E1 -5865.156,E2 -5865.156} C_VEL
LIN {X 0,Y 504.504,Z 711.748,A -85,B 0,C 180,E1 -5866.176,E2 -5866.176} C_VEL
LIN {X 0,Y 505.006,Z 699.513,A -85,B 0,C 180,E1 -5867.095,E2 -5867.095} C_VEL
LIN {X 0,Y 505.545,Z 686.227,A -85,B 0,C 180,E1 -5867.912,E2 -5867.912} C_VEL
LIN {X 0,Y 506.025,Z 672.646,A -85,B 0,C 180,E1 -5868.575,E2 -5868.575} C_VEL
LIN {X 0,Y 506.406,Z 658.801,A -85,B 0,C 180,E1 -5869.101,E2 -5869.101} C_VEL
LIN {X 0,Y 506.84,Z 642.047,A -85,B 0,C 180,E1 -5869.568,E2 -5869.568} C_VEL
LIN {X 0,Y 507.091,Z 622.57,A -85,B 0,C 180,E1 -5869.901,E2 -5869.901} C_VEL
LIN {X 0,Y 508.279,Z 486.346,A -85,B 0,C 180,E1 -5871.934,E2 -5871.934} C_VEL
LIN {X 0,Y 505.91,Z 469.554,A -85,B 0,C 180,E1 -5872.318,E2 -5872.318} C_VEL
LIN {X 0,Y 506.914,Z 439.552,A -85,B 0,C 180,E1 -5875.233,E2 -5875.233} C_VEL
LIN {X 0,Y 508.116,Z 407.63,A -85,B 0,C 180,E1 -5878.387,E2 -5878.387} C_VEL
LIN {X 0,Y 508.864,Z 390.169,A -85,B 0,C 180,E1 -5880.151,E2 -5880.151} C_VEL
LIN {X 0,Y 505.375,Z 377.387,A -85,B 0,C 180,E1 -5881.692,E2 -5881.692} C_VEL
LIN {X 0,Y 502.812,Z 368.663,A -85,B 0,C 180,E1 -5882.809,E2 -5882.809} C_VEL
LIN {X 0,Y 502.741,Z 368.486,A -85,B 0,C 180,E1 -5885.826,E2 -5885.826} C_VEL
LIN {X 0,Y 502.772,Z 368.482,A -85,B 0,C 180,E1 -5888.977,E2 -5888.977} C_VEL
LIN {X 0,Y 502.76,Z 368.488,A -85,B 0,C 180,E1 -5892.194,E2 -5892.194} C_VEL
LIN {X 0,Y 502.765,Z 368.48,A -85,B 0,C 180,E1 -5895.47,E2 -5895.47} C_VEL
LIN {X 0,Y 502.749,Z 368.478,A -85,B 0,C 180,E1 -5898.927,E2 -5898.927} C_VEL
LIN {X 0,Y 502.745,Z 368.486,A -85,B 0,C 180,E1 -5902.042,E2 -5902.042} C_VEL
LIN {X 0,Y 502.768,Z 368.463,A -85,B 0,C 180,E1 -5905.032,E2 -5905.032} C_VEL
LIN {X 0,Y 502.767,Z 368.479,A -85,B 0,C 180,E1 -5907.914,E2 -5907.914} C_VEL
LIN {X 0,Y 502.789,Z 368.477,A -85,B 0,C 180,E1 -5910.71,E2 -5910.71} C_VEL
LIN {X 0,Y 502.767,Z 368.479,A -85,B 0,C 180,E1 -5913.457,E2 -5913.457} C_VEL
LIN {X 0,Y 502.75,Z 368.479,A -85,B 0,C 180,E1 -5916.084,E2 -5916.084} C_VEL
LIN {X 0,Y 502.761,Z 368.481,A -85,B 0,C 180,E1 -5918.688,E2 -5918.688} C_VEL
LIN {X 0,Y 502.79,Z 368.475,A -85,B 0,C 180,E1 -5921.247,E2 -5921.247} C_VEL
LIN {X 0,Y 502.818,Z 368.471,A -85,B 0,C 180,E1 -5924.664,E2 -5924.664} C_VEL
LIN {X 0,Y 502.86,Z 368.47,A -85,B 0,C 180,E1 -5928.039,E2 -5928.039} C_VEL
LIN {X 0,Y 502.823,Z 368.47,A -85,B 0,C 180,E1 -5931.156,E2 -5931.156} C_VEL
LIN {X 0,Y 502.832,Z 368.47,A -85,B 0,C 180,E1 -5933.58,E2 -5933.58} C_VEL
LIN {X 0,Y 502.848,Z 368.473,A -85,B 0,C 180,E1 -5936.795,E2 -5936.795} C_VEL
LIN {X 0,Y 502.884,Z 368.47,A -85,B 0,C 180,E1 -5938.398,E2 -5938.398} C_VEL
LIN {X 0,Y 502.993,Z 368.448,A -85,B 0,C 180,E1 -5940.801,E2 -5940.801} C_VEL
LIN {X 0,Y 502.994,Z 368.45,A -85,B 0,C 180,E1 -5942.402,E2 -5942.402} C_VEL
LIN {X 0,Y 502.902,Z 368.459,A -85,B 0,C 180,E1 -5945.614,E2 -5945.614} C_VEL
LIN {X 0,Y 502.855,Z 368.466,A -85,B 0,C 180,E1 -5948.034,E2 -5948.034} C_VEL
LIN {X 0,Y 502.856,Z 368.461,A -85,B 0,C 180,E1 -5951.284,E2 -5951.284} C_VEL
LIN {X 0,Y 502.815,Z 368.48,A -85,B 0,C 180,E1 -5954.572,E2 -5954.572} C_VEL
LIN {X 0,Y 502.796,Z 368.476,A -85,B 0,C 180,E1 -5957.07,E2 -5957.07} C_VEL
LIN {X 0,Y 502.803,Z 368.473,A -85,B 0,C 180,E1 -5959.601,E2 -5959.601} C_VEL
LIN {X 0,Y 502.787,Z 368.482,A -85,B 0,C 180,E1 -5962.703,E2 -5962.703} C_VEL
LIN {X 0,Y 502.753,Z 368.476,A -85,B 0,C 180,E1 -5965.68,E2 -5965.68} C_VEL
LIN {X 0,Y 502.757,Z 368.485,A -85,B 0,C 180,E1 -5968.378,E2 -5968.378} C_VEL
LIN {X 0,Y 502.751,Z 368.485,A -85,B 0,C 180,E1 -5971.146,E2 -5971.146} C_VEL
LIN {X 0,Y 502.775,Z 368.48,A -85,B 0,C 180,E1 -5973.996,E2 -5973.996} C_VEL
LIN {X 0,Y 502.739,Z 368.472,A -85,B 0,C 180,E1 -5977.175,E2 -5977.175} C_VEL
LIN {X 0,Y 502.757,Z 368.482,A -85,B 0,C 180,E1 -5980.018,E2 -5980.018} C_VEL
LIN {X 0,Y 502.727,Z 368.483,A -85,B 0,C 180,E1 -5983.236,E2 -5983.236} C_VEL
LIN {X 0,Y 502.755,Z 368.48,A -85,B 0,C 180,E1 -5985.66,E2 -5985.66} C_VEL
LIN {X 0,Y 502.752,Z 368.484,A -85,B 0,C 180,E1 -5989.014,E2 -5989.014} C_VEL
LIN {X 0,Y 502.751,Z 368.485,A -85,B 0,C 180,E1 -5992.044,E2 -5992.044} C_VEL
LIN {X 0,Y 502.774,Z 368.472,A -85,B 0,C 180,E1 -5995.034,E2 -5995.034} C_VEL
LIN {X 0,Y 502.783,Z 368.453,A -85,B 0,C 180,E1 -5996.027,E2 -5996.027} C_VEL
LIN {X 0,Y 502.732,Z 369.359,A -85,B 0,C 180,E1 -5996.367,E2 -5996.367} C_VEL
LIN {X 0,Y 502.406,Z 372.914,A -85,B 0,C 180,E1 -5996.836,E2 -5996.836} C_VEL
LIN {X 0,Y 501.154,Z 386.21,A -85,B 0,C 180,E1 -5998.184,E2 -5998.184} C_VEL
LIN {X 0,Y 501.666,Z 390.083,A -85,B 0,C 180,E1 -5998.653,E2 -5998.653} C_VEL
LIN {X 0,Y 502.132,Z 392.524,A -85,B 0,C 180,E1 -5998.946,E2 -5998.946} C_VEL
LIN {X 0,Y 501.038,Z 423.308,A -85,B 0,C 180,E1 -6002.242,E2 -6002.242} C_VEL
LIN {X 0,Y 499.943,Z 454.372,A -85,B 0,C 180,E1 -6005.501,E2 -6005.501} C_VEL
LIN {X 0,Y 499.46,Z 472.424,A -85,B 0,C 180,E1 -6007.31,E2 -6007.31} C_VEL
LIN {X 0,Y 502.189,Z 489.163,A -85,B 0,C 180,E1 -6007.719,E2 -6007.719} C_VEL
LIN {X 0,Y 500.795,Z 640.445,A -85,B 0,C 180,E1 -6009.958,E2 -6009.958} C_VEL
LIN {X 0,Y 500.425,Z 656.268,A -85,B 0,C 180,E1 -6010.353,E2 -6010.353} C_VEL
LIN {X 0,Y 499.944,Z 670.7,A -85,B 0,C 180,E1 -6010.875,E2 -6010.875} C_VEL
LIN {X 0,Y 499.372,Z 684.654,A -85,B 0,C 180,E1 -6011.541,E2 -6011.541} C_VEL
LIN {X 0,Y 498.767,Z 698.369,A -85,B 0,C 180,E1 -6012.367,E2 -6012.367} C_VEL
LIN {X 0,Y 498.15,Z 710.979,A -85,B 0,C 180,E1 -6013.296,E2 -6013.296} C_VEL
LIN {X 0,Y 497.465,Z 723.715,A -85,B 0,C 180,E1 -6014.431,E2 -6014.431} C_VEL
LIN {X 0,Y 496.805,Z 735.266,A -85,B 0,C 180,E1 -6015.668,E2 -6015.668} C_VEL
LIN {X 0,Y 496.325,Z 745.003,A -85,B 0,C 180,E1 -6016.907,E2 -6016.907} C_VEL
LIN {X 0,Y 495.909,Z 754.142,A -85,B 0,C 180,E1 -6018.284,E2 -6018.284} C_VEL
LIN {X 0,Y 495.551,Z 762.473,A -85,B 0,C 180,E1 -6019.79,E2 -6019.79} C_VEL
LIN {X 0,Y 495.311,Z 769.878,A -85,B 0,C 180,E1 -6021.433,E2 -6021.433} C_VEL
LIN {X 0,Y 495.115,Z 775.76,A -85,B 0,C 180,E1 -6023.071,E2 -6023.071} C_VEL
LIN {X 0,Y 495.106,Z 779.23,A -85,B 0,C 180,E1 -6024.299,E2 -6024.299} C_VEL
LIN {X 0,Y 494.993,Z 782.768,A -85,B 0,C 180,E1 -6025.93,E2 -6025.93} C_VEL
LIN {X 0,Y 494.971,Z 785.11,A -85,B 0,C 180,E1 -6027.56,E2 -6027.56} C_VEL
LIN {X 0,Y 494.907,Z 786.305,A -85,B 0,C 180,E1 -6029.188,E2 -6029.188} C_VEL
LIN {X 0,Y 494.908,Z 786.323,A -85,B 0,C 180,E1 -6030.815,E2 -6030.815} C_VEL
LIN {X 0,Y 494.972,Z 785.199,A -85,B 0,C 180,E1 -6032.443,E2 -6032.443} C_VEL
LIN {X 0,Y 494.993,Z 782.927,A -85,B 0,C 180,E1 -6034.072,E2 -6034.072} C_VEL
LIN {X 0,Y 495.098,Z 779.454,A -85,B 0,C 180,E1 -6035.704,E2 -6035.704} C_VEL
LIN {X 0,Y 495.167,Z 774.7,A -85,B 0,C 180,E1 -6037.34,E2 -6037.34} C_VEL
LIN {X 0,Y 495.337,Z 768.544,A -85,B 0,C 180,E1 -6038.98,E2 -6038.98} C_VEL
LIN {X 0,Y 495.708,Z 760.801,A -85,B 0,C 180,E1 -6040.622,E2 -6040.622} C_VEL
LIN {X 0,Y 495.994,Z 752.171,A -85,B 0,C 180,E1 -6042.123,E2 -6042.123} C_VEL
LIN {X 0,Y 496.489,Z 742.601,A -85,B 0,C 180,E1 -6043.508,E2 -6043.508} C_VEL
LIN {X 0,Y 496.984,Z 732.456,A -85,B 0,C 180,E1 -6044.748,E2 -6044.748} C_VEL
LIN {X 0,Y 497.64,Z 720.656,A -85,B 0,C 180,E1 -6045.955,E2 -6045.955} C_VEL
LIN {X 0,Y 498.264,Z 708.194,A -85,B 0,C 180,E1 -6047.019,E2 -6047.019} C_VEL
LIN {X 0,Y 498.982,Z 695.004,A -85,B 0,C 180,E1 -6047.946,E2 -6047.946} C_VEL
LIN {X 0,Y 499.519,Z 681.437,A -85,B 0,C 180,E1 -6048.722,E2 -6048.722} C_VEL
LIN {X 0,Y 500.097,Z 666.666,A -85,B 0,C 180,E1 -6049.381,E2 -6049.381} C_VEL
LIN {X 0,Y 500.546,Z 651.549,A -85,B 0,C 180,E1 -6049.878,E2 -6049.878} C_VEL
LIN {X 0,Y 500.877,Z 636.015,A -85,B 0,C 180,E1 -6050.214,E2 -6050.214} C_VEL
LIN {X 0,Y 502.155,Z 488.666,A -85,B 0,C 180,E1 -6052.38,E2 -6052.38} C_VEL
LIN {X 0,Y 499.489,Z 472.761,A -85,B 0,C 180,E1 -6052.761,E2 -6052.761} C_VEL
LIN {X 0,Y 500.062,Z 449.945,A -85,B 0,C 180,E1 -6055.049,E2 -6055.049} C_VEL
LIN {X 0,Y 501.1,Z 420.869,A -85,B 0,C 180,E1 -6058.112,E2 -6058.112} C_VEL
LIN {X 0,Y 502.138,Z 393.044,A -85,B 0,C 180,E1 -6061.092,E2 -6061.092} C_VEL
LIN {X 0,Y 501.043,Z 387.655,A -85,B 0,C 180,E1 -6061.748,E2 -6061.748} C_VEL
LIN {X 0,Y 496.434,Z 371.949,A -85,B 0,C 180,E1 -6063.74,E2 -6063.74} C_VEL
LIN {X 0,Y 495.714,Z 369.539,A -85,B 0,C 180,E1 -6064.088,E2 -6064.088} C_VEL
LIN {X 0,Y 495.691,Z 369.368,A -85,B 0,C 180,E1 -6067.566,E2 -6067.566} C_VEL
LIN {X 0,Y 495.709,Z 369.361,A -85,B 0,C 180,E1 -6070.04,E2 -6070.04} C_VEL
LIN {X 0,Y 495.693,Z 369.359,A -85,B 0,C 180,E1 -6072.888,E2 -6072.888} C_VEL
LIN {X 0,Y 495.716,Z 369.353,A -85,B 0,C 180,E1 -6075.997,E2 -6075.997} C_VEL
LIN {X 0,Y 495.713,Z 369.352,A -85,B 0,C 180,E1 -6079.295,E2 -6079.295} C_VEL
LIN {X 0,Y 495.718,Z 369.361,A -85,B 0,C 180,E1 -6081.405,E2 -6081.405} C_VEL
LIN {X 0,Y 495.731,Z 369.351,A -85,B 0,C 180,E1 -6084.461,E2 -6084.461} C_VEL
LIN {X 0,Y 495.728,Z 369.362,A -85,B 0,C 180,E1 -6087.403,E2 -6087.403} C_VEL
LIN {X 0,Y 495.742,Z 369.355,A -85,B 0,C 180,E1 -6090.252,E2 -6090.252} C_VEL
LIN {X 0,Y 495.725,Z 369.363,A -85,B 0,C 180,E1 -6093.275,E2 -6093.275} C_VEL
LIN {X 0,Y 495.707,Z 369.363,A -85,B 0,C 180,E1 -6095.723,E2 -6095.723} C_VEL
LIN {X 0,Y 495.796,Z 369.533,A -85,B 0,C 180,E1 -6098.592,E2 -6098.592} C_VEL
LIN {X 0,Y 497.408,Z 377.76,A -85,B 0,C 180,E1 -6100.178,E2 -6100.178} C_VEL
LIN {X 0,Y 497.656,Z 380.425,A -85,B 0,C 180,E1 -6100.603,E2 -6100.603} C_VEL
LIN {X 0,Y 500.409,Z 392.44,A -85,B 0,C 180,E1 -6100.937,E2 -6100.937} C_VEL
LIN {X 0,Y 499.114,Z 519.164,A -85,B 0,C 180,E1 -6102.961,E2 -6102.961} C_VEL
LIN {X 0,Y 498.944,Z 533.122,A -85,B 0,C 180,E1 -6103.343,E2 -6103.343} C_VEL
LIN {X 0,Y 498.679,Z 547.105,A -85,B 0,C 180,E1 -6103.891,E2 -6103.891} C_VEL
LIN {X 0,Y 498.365,Z 560.074,A -85,B 0,C 180,E1 -6104.563,E2 -6104.563} C_VEL
LIN {X 0,Y 497.977,Z 571.249,A -85,B 0,C 180,E1 -6105.283,E2 -6105.283} C_VEL
LIN {X 0,Y 497.578,Z 583.001,A -85,B 0,C 180,E1 -6106.211,E2 -6106.211} C_VEL
LIN {X 0,Y 497.137,Z 594.147,A -85,B 0,C 180,E1 -6107.28,E2 -6107.28} C_VEL
LIN {X 0,Y 496.839,Z 603.571,A -85,B 0,C 180,E1 -6108.371,E2 -6108.371} C_VEL
LIN {X 0,Y 496.42,Z 612.472,A -85,B 0,C 180,E1 -6109.601,E2 -6109.601} C_VEL
LIN {X 0,Y 496.093,Z 620.979,A -85,B 0,C 180,E1 -6111.035,E2 -6111.035} C_VEL
LIN {X 0,Y 495.896,Z 626.899,A -85,B 0,C 180,E1 -6112.262,E2 -6112.262} C_VEL
LIN {X 0,Y 495.783,Z 631.774,A -85,B 0,C 180,E1 -6113.488,E2 -6113.488} C_VEL
LIN {X 0,Y 495.538,Z 636.844,A -85,B 0,C 180,E1 -6115.118,E2 -6115.118} C_VEL
LIN {X 0,Y 495.46,Z 640.409,A -85,B 0,C 180,E1 -6116.747,E2 -6116.747} C_VEL
LIN {X 0,Y 495.395,Z 642.584,A -85,B 0,C 180,E1 -6118.374,E2 -6118.374} C_VEL
LIN {X 0,Y 495.438,Z 643.412,A -85,B 0,C 180,E1 -6120,E2 -6120} C_VEL
LIN {X 0,Y 495.395,Z 642.919,A -85,B 0,C 180,E1 -6121.626,E2 -6121.626} C_VEL
LIN {X 0,Y 495.528,Z 641.061,A -85,B 0,C 180,E1 -6123.252,E2 -6123.252} C_VEL
LIN {X 0,Y 495.614,Z 637.831,A -85,B 0,C 180,E1 -6124.881,E2 -6124.881} C_VEL
LIN {X 0,Y 495.905,Z 633.087,A -85,B 0,C 180,E1 -6126.51,E2 -6126.51} C_VEL
LIN {X 0,Y 495.998,Z 628.477,A -85,B 0,C 180,E1 -6127.736,E2 -6127.736} C_VEL
LIN {X 0,Y 496.283,Z 621.737,A -85,B 0,C 180,E1 -6129.167,E2 -6129.167} C_VEL
LIN {X 0,Y 496.619,Z 613.326,A -85,B 0,C 180,E1 -6130.601,E2 -6130.601} C_VEL
LIN {X 0,Y 497.072,Z 604.454,A -85,B 0,C 180,E1 -6131.83,E2 -6131.83} C_VEL
LIN {X 0,Y 497.462,Z 595.321,A -85,B 0,C 180,E1 -6132.885,E2 -6132.885} C_VEL
LIN {X 0,Y 497.862,Z 583.808,A -85,B 0,C 180,E1 -6133.989,E2 -6133.989} C_VEL
LIN {X 0,Y 498.196,Z 571.949,A -85,B 0,C 180,E1 -6134.919,E2 -6134.919} C_VEL
LIN {X 0,Y 498.622,Z 558.651,A -85,B 0,C 180,E1 -6135.743,E2 -6135.743} C_VEL
LIN {X 0,Y 498.951,Z 544.791,A -85,B 0,C 180,E1 -6136.407,E2 -6136.407} C_VEL
LIN {X 0,Y 499.165,Z 530.121,A -85,B 0,C 180,E1 -6136.921,E2 -6136.921} C_VEL
LIN {X 0,Y 499.33,Z 515.964,A -85,B 0,C 180,E1 -6137.245,E2 -6137.245} C_VEL
LIN {X 0,Y 500.698,Z 422.76,A -85,B 0,C 180,E1 -6138.851,E2 -6138.851} C_VEL
LIN {X 0,Y 501.24,Z 393.306,A -85,B 0,C 180,E1 -6139.388,E2 -6139.388} C_VEL
LIN {X 0,Y 499.187,Z 385.888,A -85,B 0,C 180,E1 -6139.661,E2 -6139.661} C_VEL
LIN {X 0,Y 499.065,Z 383.04,A -85,B 0,C 180,E1 -6140.183,E2 -6140.183} C_VEL
LIN {X 0,Y 497.121,Z 374.769,A -85,B 0,C 180,E1 -6142.002,E2 -6142.002} C_VEL
LIN {X 0,Y 495.753,Z 369.414,A -85,B 0,C 180,E1 -6143.27,E2 -6143.27} C_VEL
LIN {X 0,Y 495.796,Z 369.354,A -85,B 0,C 180,E1 -6146.068,E2 -6146.068} C_VEL
LIN {X 0,Y 495.777,Z 369.357,A -85,B 0,C 180,E1 -6148.814,E2 -6148.814} C_VEL
LIN {X 0,Y 495.76,Z 369.356,A -85,B 0,C 180,E1 -6151.725,E2 -6151.725} C_VEL
LIN {X 0,Y 495.772,Z 369.358,A -85,B 0,C 180,E1 -6154.693,E2 -6154.693} C_VEL
LIN {X 0,Y 495.725,Z 369.359,A -85,B 0,C 180,E1 -6157.562,E2 -6157.562} C_VEL
LIN {X 0,Y 495.762,Z 369.358,A -85,B 0,C 180,E1 -6160.046,E2 -6160.046} C_VEL
LIN {X 0,Y 495.719,Z 369.361,A -85,B 0,C 180,E1 -6162.884,E2 -6162.884} C_VEL
LIN {X 0,Y 495.727,Z 369.363,A -85,B 0,C 180,E1 -6165.997,E2 -6165.997} C_VEL
LIN {X 0,Y 495.733,Z 369.36,A -85,B 0,C 180,E1 -6169.296,E2 -6169.296} C_VEL
LIN {X 0,Y 495.727,Z 369.361,A -85,B 0,C 180,E1 -6171.405,E2 -6171.405} C_VEL
LIN {X 0,Y 495.73,Z 369.362,A -85,B 0,C 180,E1 -6174.46,E2 -6174.46} C_VEL
LIN {X 0,Y 495.77,Z 369.552,A -85,B 0,C 180,E1 -6176.877,E2 -6176.877} C_VEL
LIN {X 0,Y 498.718,Z 379.266,A -85,B 0,C 180,E1 -6178.282,E2 -6178.282} C_VEL
LIN {X 0,Y 501.508,Z 390.272,A -85,B 0,C 180,E1 -6179.701,E2 -6179.701} C_VEL
LIN {X 0,Y 501.158,Z 402.014,A -85,B 0,C 180,E1 -6180.95,E2 -6180.95} C_VEL
LIN {X 0,Y 499.782,Z 433.428,A -85,B 0,C 180,E1 -6184.155,E2 -6184.155} C_VEL
LIN {X 0,Y 498.821,Z 462.133,A -85,B 0,C 180,E1 -6186.984,E2 -6186.984} C_VEL
LIN {X 0,Y 498.725,Z 466.71,A -85,B 0,C 180,E1 -6187.39,E2 -6187.39} C_VEL
LIN {X 0,Y 501.485,Z 488.03,A -85,B 0,C 180,E1 -6187.882,E2 -6187.882} C_VEL
LIN {X 0,Y 500.147,Z 640.827,A -85,B 0,C 180,E1 -6190.156,E2 -6190.156} C_VEL
LIN {X 0,Y 499.826,Z 656.483,A -85,B 0,C 180,E1 -6190.554,E2 -6190.554} C_VEL
LIN {X 0,Y 499.371,Z 671.582,A -85,B 0,C 180,E1 -6191.112,E2 -6191.112} C_VEL
LIN {X 0,Y 498.838,Z 686.242,A -85,B 0,C 180,E1 -6191.836,E2 -6191.836} C_VEL
LIN {X 0,Y 498.203,Z 699.521,A -85,B 0,C 180,E1 -6192.661,E2 -6192.661} C_VEL
LIN {X 0,Y 497.586,Z 713.259,A -85,B 0,C 180,E1 -6193.72,E2 -6193.72} C_VEL
LIN {X 0,Y 497.012,Z 725.201,A -85,B 0,C 180,E1 -6194.834,E2 -6194.834} C_VEL
LIN {X 0,Y 496.511,Z 736.32,A -85,B 0,C 180,E1 -6196.075,E2 -6196.075} C_VEL
LIN {X 0,Y 496.017,Z 747.079,A -85,B 0,C 180,E1 -6197.52,E2 -6197.52} C_VEL
LIN {X 0,Y 495.686,Z 756.014,A -85,B 0,C 180,E1 -6198.964,E2 -6198.964} C_VEL
LIN {X 0,Y 495.379,Z 764.355,A -85,B 0,C 180,E1 -6200.609,E2 -6200.609} C_VEL
LIN {X 0,Y 495.221,Z 771.031,A -85,B 0,C 180,E1 -6202.251,E2 -6202.251} C_VEL
LIN {X 0,Y 495.146,Z 775.825,A -85,B 0,C 180,E1 -6203.733,E2 -6203.733} C_VEL
LIN {X 0,Y 495.063,Z 779.249,A -85,B 0,C 180,E1 -6205.113,E2 -6205.113} C_VEL
LIN {X 0,Y 495.083,Z 782.185,A -85,B 0,C 180,E1 -6206.744,E2 -6206.744} C_VEL
LIN {X 0,Y 495.015,Z 783.936,A -85,B 0,C 180,E1 -6208.372,E2 -6208.372} C_VEL
LIN {X 0,Y 494.973,Z 784.534,A -85,B 0,C 180,E1 -6209.999,E2 -6209.999} C_VEL
LIN {X 0,Y 495.014,Z 783.937,A -85,B 0,C 180,E1 -6211.626,E2 -6211.626} C_VEL
LIN {X 0,Y 495.091,Z 782.186,A -85,B 0,C 180,E1 -6213.254,E2 -6213.254} C_VEL
LIN {X 0,Y 495.058,Z 779.25,A -85,B 0,C 180,E1 -6214.885,E2 -6214.885} C_VEL
LIN {X 0,Y 495.123,Z 775.062,A -85,B 0,C 180,E1 -6216.519,E2 -6216.519} C_VEL
LIN {X 0,Y 495.261,Z 769.507,A -85,B 0,C 180,E1 -6218.157,E2 -6218.157} C_VEL
LIN {X 0,Y 495.418,Z 762.424,A -85,B 0,C 180,E1 -6219.8,E2 -6219.8} C_VEL
LIN {X 0,Y 495.742,Z 754.834,A -85,B 0,C 180,E1 -6221.239,E2 -6221.239} C_VEL
LIN {X 0,Y 495.997,Z 747.097,A -85,B 0,C 180,E1 -6222.478,E2 -6222.478} C_VEL
LIN {X 0,Y 496.479,Z 736.34,A -85,B 0,C 180,E1 -6223.923,E2 -6223.923} C_VEL
LIN {X 0,Y 497.022,Z 724.205,A -85,B 0,C 180,E1 -6225.268,E2 -6225.268} C_VEL
LIN {X 0,Y 497.672,Z 711.784,A -85,B 0,C 180,E1 -6226.404,E2 -6226.404} C_VEL
LIN {X 0,Y 498.249,Z 697.992,A -85,B 0,C 180,E1 -6227.44,E2 -6227.44} C_VEL
LIN {X 0,Y 498.826,Z 684.365,A -85,B 0,C 180,E1 -6228.268,E2 -6228.268} C_VEL
LIN {X 0,Y 499.339,Z 671.651,A -85,B 0,C 180,E1 -6228.886,E2 -6228.886} C_VEL
LIN {X 0,Y 499.77,Z 656.499,A -85,B 0,C 180,E1 -6229.449,E2 -6229.449} C_VEL
LIN {X 0,Y 500.128,Z 640.986,A -85,B 0,C 180,E1 -6229.842,E2 -6229.842} C_VEL
LIN {X 0,Y 501.65,Z 488.412,A -85,B 0,C 180,E1 -6232.173,E2 -6232.173} C_VEL
LIN {X 0,Y 499.079,Z 469.071,A -85,B 0,C 180,E1 -6232.617,E2 -6232.617} C_VEL
LIN {X 0,Y 500.136,Z 439.911,A -85,B 0,C 180,E1 -6235.488,E2 -6235.488} C_VEL
LIN {X 0,Y 501.394,Z 409.202,A -85,B 0,C 180,E1 -6238.574,E2 -6238.574} C_VEL
LIN {X 0,Y 502.181,Z 392.755,A -85,B 0,C 180,E1 -6240.251,E2 -6240.251} C_VEL
LIN {X 0,Y 500.861,Z 386.976,A -85,B 0,C 180,E1 -6240.939,E2 -6240.939} C_VEL
LIN {X 0,Y 495.762,Z 369.533,A -85,B 0,C 180,E1 -6243.162,E2 -6243.162} C_VEL
LIN {X 0,Y 495.718,Z 369.36,A -85,B 0,C 180,E1 -6245.538,E2 -6245.538} C_VEL
LIN {X 0,Y 495.729,Z 369.361,A -85,B 0,C 180,E1 -6248.763,E2 -6248.763} C_VEL
LIN {X 0,Y 495.714,Z 369.361,A -85,B 0,C 180,E1 -6251.783,E2 -6251.783} C_VEL
LIN {X 0,Y 495.721,Z 369.357,A -85,B 0,C 180,E1 -6255.14,E2 -6255.14} C_VEL
LIN {X 0,Y 495.71,Z 369.345,A -85,B 0,C 180,E1 -6258.214,E2 -6258.214} C_VEL
LIN {X 0,Y 495.725,Z 369.357,A -85,B 0,C 180,E1 -6261.234,E2 -6261.234} C_VEL
LIN {X 0,Y 495.714,Z 369.341,A -85,B 0,C 180,E1 -6264.46,E2 -6264.46} C_VEL
LIN {X 0,Y 495.737,Z 369.352,A -85,B 0,C 180,E1 -6267.403,E2 -6267.403} C_VEL
LIN {X 0,Y 495.742,Z 369.357,A -85,B 0,C 180,E1 -6270.252,E2 -6270.252} C_VEL
LIN {X 0,Y 495.726,Z 369.356,A -85,B 0,C 180,E1 -6273.269,E2 -6273.269} C_VEL
LIN {X 0,Y 495.722,Z 369.363,A -85,B 0,C 180,E1 -6276.612,E2 -6276.612} C_VEL
LIN {X 0,Y 495.763,Z 369.347,A -85,B 0,C 180,E1 -6279.324,E2 -6279.324} C_VEL
LIN {X 0,Y 495.763,Z 369.351,A -85,B 0,C 180,E1 -6281.828,E2 -6281.828} C_VEL
LIN {X 0,Y 495.759,Z 369.346,A -85,B 0,C 180,E1 -6285.216,E2 -6285.216} C_VEL
LIN {X 0,Y 495.831,Z 369.347,A -85,B 0,C 180,E1 -6288.554,E2 -6288.554} C_VEL
LIN {X 0,Y 495.795,Z 369.345,A -85,B 0,C 180,E1 -6291.851,E2 -6291.851} C_VEL
LIN {X 0,Y 495.797,Z 369.341,A -85,B 0,C 180,E1 -6295.121,E2 -6295.121} C_VEL
LIN {X 0,Y 495.963,Z 369.325,A -85,B 0,C 180,E1 -6297.564,E2 -6297.564} C_VEL
LIN {X 0,Y 495.944,Z 369.326,A -85,B 0,C 180,E1 -6300.812,E2 -6300.812} C_VEL
LIN {X 0,Y 495.962,Z 369.326,A -85,B 0,C 180,E1 -6302.437,E2 -6302.437} C_VEL
LIN {X 0,Y 495.858,Z 369.336,A -85,B 0,C 180,E1 -6305.694,E2 -6305.694} C_VEL
LIN {X 0,Y 495.812,Z 369.344,A -85,B 0,C 180,E1 -6308.149,E2 -6308.149} C_VEL
LIN {X 0,Y 495.832,Z 369.335,A -85,B 0,C 180,E1 -6311.446,E2 -6311.446} C_VEL
LIN {X 0,Y 495.764,Z 369.355,A -85,B 0,C 180,E1 -6314.784,E2 -6314.784} C_VEL
LIN {X 0,Y 495.741,Z 369.352,A -85,B 0,C 180,E1 -6317.32,E2 -6317.32} C_VEL
LIN {X 0,Y 495.752,Z 369.352,A -85,B 0,C 180,E1 -6319.891,E2 -6319.891} C_VEL
LIN {X 0,Y 495.743,Z 369.361,A -85,B 0,C 180,E1 -6322.861,E2 -6322.861} C_VEL
LIN {X 0,Y 495.696,Z 369.357,A -85,B 0,C 180,E1 -6326.073,E2 -6326.073} C_VEL
LIN {X 0,Y 495.706,Z 369.361,A -85,B 0,C 180,E1 -6328.819,E2 -6328.819} C_VEL
LIN {X 0,Y 495.723,Z 369.357,A -85,B 0,C 180,E1 -6331.723,E2 -6331.723} C_VEL
LIN {X 0,Y 495.747,Z 369.363,A -85,B 0,C 180,E1 -6334.694,E2 -6334.694} C_VEL
LIN {X 0,Y 495.694,Z 369.348,A -85,B 0,C 180,E1 -6337.565,E2 -6337.565} C_VEL
LIN {X 0,Y 495.73,Z 369.357,A -85,B 0,C 180,E1 -6340.046,E2 -6340.046} C_VEL
LIN {X 0,Y 495.679,Z 369.357,A -85,B 0,C 180,E1 -6342.888,E2 -6342.888} C_VEL
LIN {X 0,Y 495.702,Z 369.359,A -85,B 0,C 180,E1 -6345.998,E2 -6345.998} C_VEL
LIN {X 0,Y 495.715,Z 369.357,A -85,B 0,C 180,E1 -6349.297,E2 -6349.297} C_VEL
LIN {X 0,Y 495.713,Z 369.363,A -85,B 0,C 180,E1 -6351.407,E2 -6351.407} C_VEL
LIN {X 0,Y 495.72,Z 369.361,A -85,B 0,C 180,E1 -6354.462,E2 -6354.462} C_VEL
LIN {X 0,Y 495.788,Z 369.512,A -85,B 0,C 180,E1 -6356.006,E2 -6356.006} C_VEL
LIN {X 0,Y 497.256,Z 374.525,A -85,B 0,C 180,E1 -6356.683,E2 -6356.683} C_VEL
LIN {X 0,Y 501.666,Z 390.083,A -85,B 0,C 180,E1 -6358.653,E2 -6358.653} C_VEL
LIN {X 0,Y 501.871,Z 392.846,A -85,B 0,C 180,E1 -6358.966,E2 -6358.966} C_VEL
LIN {X 0,Y 500.875,Z 397.299,A -85,B 0,C 180,E1 -6359.392,E2 -6359.392} C_VEL
LIN {X 0,Y 495.639,Z 409.575,A -85,B 0,C 180,E1 -6360.434,E2 -6360.434} C_VEL
LIN {X 0,Y 494.7,Z 414.108,A -85,B 0,C 180,E1 -6360.883,E2 -6360.883} C_VEL
LIN {X 0,Y 493.792,Z 438.393,A -85,B 0,C 180,E1 -6363.491,E2 -6363.491} C_VEL
LIN {X 0,Y 492.89,Z 465.612,A -85,B 0,C 180,E1 -6366.324,E2 -6366.324} C_VEL
LIN {X 0,Y 492.753,Z 472.753,A -85,B 0,C 180,E1 -6367.006,E2 -6367.006} C_VEL
LIN {X 0,Y 495.621,Z 490.87,A -85,B 0,C 180,E1 -6367.436,E2 -6367.436} C_VEL
LIN {X 0,Y 494.142,Z 640.297,A -85,B 0,C 180,E1 -6369.677,E2 -6369.677} C_VEL
LIN {X 0,Y 493.752,Z 655.925,A -85,B 0,C 180,E1 -6370.068,E2 -6370.068} C_VEL
LIN {X 0,Y 493.213,Z 670.898,A -85,B 0,C 180,E1 -6370.615,E2 -6370.615} C_VEL
LIN {X 0,Y 492.619,Z 684.607,A -85,B 0,C 180,E1 -6371.278,E2 -6371.278} C_VEL
LIN {X 0,Y 491.975,Z 698.332,A -85,B 0,C 180,E1 -6372.115,E2 -6372.115} C_VEL
LIN {X 0,Y 491.291,Z 710.948,A -85,B 0,C 180,E1 -6373.056,E2 -6373.056} C_VEL
LIN {X 0,Y 490.585,Z 723.689,A -85,B 0,C 180,E1 -6374.207,E2 -6374.207} C_VEL
LIN {X 0,Y 489.888,Z 735.244,A -85,B 0,C 180,E1 -6375.461,E2 -6375.461} C_VEL
LIN {X 0,Y 489.359,Z 744.984,A -85,B 0,C 180,E1 -6376.717,E2 -6376.717} C_VEL
LIN {X 0,Y 488.9,Z 754.374,A -85,B 0,C 180,E1 -6378.157,E2 -6378.157} C_VEL
LIN {X 0,Y 488.528,Z 762.457,A -85,B 0,C 180,E1 -6379.642,E2 -6379.642} C_VEL
LIN {X 0,Y 488.236,Z 769.863,A -85,B 0,C 180,E1 -6381.308,E2 -6381.308} C_VEL
LIN {X 0,Y 488.049,Z 775.746,A -85,B 0,C 180,E1 -6382.971,E2 -6382.971} C_VEL
LIN {X 0,Y 488.02,Z 779.216,A -85,B 0,C 180,E1 -6384.216,E2 -6384.216} C_VEL
LIN {X 0,Y 487.892,Z 782.755,A -85,B 0,C 180,E1 -6385.871,E2 -6385.871} C_VEL
LIN {X 0,Y 487.883,Z 785.096,A -85,B 0,C 180,E1 -6387.524,E2 -6387.524} C_VEL
LIN {X 0,Y 487.83,Z 786.291,A -85,B 0,C 180,E1 -6389.176,E2 -6389.176} C_VEL
LIN {X 0,Y 487.831,Z 786.309,A -85,B 0,C 180,E1 -6390.827,E2 -6390.827} C_VEL
LIN {X 0,Y 487.884,Z 785.184,A -85,B 0,C 180,E1 -6392.478,E2 -6392.478} C_VEL
LIN {X 0,Y 487.892,Z 782.911,A -85,B 0,C 180,E1 -6394.131,E2 -6394.131} C_VEL
LIN {X 0,Y 487.993,Z 779.437,A -85,B 0,C 180,E1 -6395.787,E2 -6395.787} C_VEL
LIN {X 0,Y 488.093,Z 774.681,A -85,B 0,C 180,E1 -6397.447,E2 -6397.447} C_VEL
LIN {X 0,Y 488.273,Z 768.524,A -85,B 0,C 180,E1 -6399.111,E2 -6399.111} C_VEL
LIN {X 0,Y 488.662,Z 760.778,A -85,B 0,C 180,E1 -6400.777,E2 -6400.777} C_VEL
LIN {X 0,Y 488.97,Z 752.699,A -85,B 0,C 180,E1 -6402.212,E2 -6402.212} C_VEL
LIN {X 0,Y 489.425,Z 744.128,A -85,B 0,C 180,E1 -6403.495,E2 -6403.495} C_VEL
LIN {X 0,Y 490.062,Z 732.421,A -85,B 0,C 180,E1 -6404.961,E2 -6404.961} C_VEL
LIN {X 0,Y 490.775,Z 720.219,A -85,B 0,C 180,E1 -6406.221,E2 -6406.221} C_VEL
LIN {X 0,Y 491.43,Z 708.144,A -85,B 0,C 180,E1 -6407.263,E2 -6407.263} C_VEL
LIN {X 0,Y 492.195,Z 694.942,A -85,B 0,C 180,E1 -6408.202,E2 -6408.202} C_VEL
LIN {X 0,Y 492.782,Z 681.362,A -85,B 0,C 180,E1 -6408.988,E2 -6408.988} C_VEL
LIN {X 0,Y 493.4,Z 666.116,A -85,B 0,C 180,E1 -6409.672,E2 -6409.672} C_VEL
LIN {X 0,Y 493.885,Z 651.396,A -85,B 0,C 180,E1 -6410.157,E2 -6410.157} C_VEL
LIN {X 0,Y 494.212,Z 635.745,A -85,B 0,C 180,E1 -6410.499,E2 -6410.499} C_VEL
LIN {X 0,Y 495.642,Z 490.162,A -85,B 0,C 180,E1 -6412.665,E2 -6412.665} C_VEL
LIN {X 0,Y 492.724,Z 472.78,A -85,B 0,C 180,E1 -6413.083,E2 -6413.083} C_VEL
LIN {X 0,Y 492.975,Z 461.753,A -85,B 0,C 180,E1 -6414.16,E2 -6414.16} C_VEL
LIN {X 0,Y 494.012,Z 432.847,A -85,B 0,C 180,E1 -6417.196,E2 -6417.196} C_VEL
LIN {X 0,Y 495.199,Z 402.388,A -85,B 0,C 180,E1 -6420.474,E2 -6420.474} C_VEL
LIN {X 0,Y 495.484,Z 394.473,A -85,B 0,C 180,E1 -6421.332,E2 -6421.332} C_VEL
LIN {X 0,Y 491.63,Z 380.11,A -85,B 0,C 180,E1 -6423.161,E2 -6423.161} C_VEL
LIN {X 0,Y 488.689,Z 370.465,A -85,B 0,C 180,E1 -6424.444,E2 -6424.444} C_VEL
